(* CoDeSys 2.3 project: WOORI_YANG_BLOCKLIFT_v0.1.pro *)
(* Libraries: INEXT_Library_V01_06.lib 6.7.18 18:58:54, lib_mat.lib 6.7.18 18:58:54, Util.lib 13.6.14 19:20:40, STANDARD_V02_00.lib 6.7.18 18:58:54, BODAS_RC28-14_30_Family_V01_03.lib 6.7.18 18:58:54, CIA405_Library_V02_01.lib 6.7.18 18:58:54, RCE_Library_V01_03.lib 6.7.18 18:58:54, OUTEXT_Library_V01_04.lib 6.7.18 18:58:54, RCE_InitParameter_V01_03.lib 6.7.18 18:58:54, BODAS-design_Library_V20.lib 6.7.18 18:58:54 *)

(* Global variable list: Global_Constant *)
VAR_GLOBAL CONSTANT
	CYCLE_DS16											: INT	  := 20;		(* [ms] main task cycle *)
END_VAR

(* Global variable list: Global_Variables *)
VAR_GLOBAL

	err_s					: applError_ts;		(* BODAS-service error structure, automatically generated by .xls *)
	para_s				: para_ts;				(* BODAS-service parameter structure, automatically generated by .xls *)
	Para					: para_ts;				(* structure for the storage of the parameter *)
	Can		  				: Can_ts;				(* structure for the CAN bus management *)
(*	Err		  				: Error_ts;				(* structure for the error management *) *)
	in_as					: in_as_ts;
(*	Input_raw			: Input_raw_ts;	(* structure for INPUT raw data *) *)
	IO_Chnl				: IO_Chnl_ts; 		(* structure for the channels of the inputs and the outputs *)

END_VAR

(* Data type in Autocode/Enums *)
TYPE applError_e:
(*********************************************)
(*  DON'T MAKE ANY CHANGES TO THIS ENUMS!!   *)
(*     FILE WAS AUTOMATICALLY GENERATED!!    *)
(*********************************************)
(

   ERR_battery_voltage_e                := 16#8000,
   ERR_central_switch_e                 := 16#8001,
   ERR_vss1_5v_e                        := 16#8002,
   ERR_sol1_A_e                         := 16#8003,
   ERR_sol1_B_e                         := 16#8004,
   ERR_can_1_e                          := 16#8005,
   ERR_joy1_ana_e                       := 16#8006

);
END_TYPE

(* Data type in Autocode/Structures *)
TYPE applError_ts:
(***********************************************)
(*  DON'T MAKE ANY CHANGES TO THIS STRUCTURE!! *)
(*      FILE WAS AUTOMATICALLY GENERATED!!     *)
(***********************************************)
STRUCT

   battery_voltage_u8               : BOOL;
   central_switch_u8                : BOOL;
   vss1_5v_u8                       : BOOL;
   sol1_a_u8                        : BOOL;
   sol1_b_u8                        : BOOL;
   can_1_u8                         : BOOL;
   joy1_ana_u8                      : BOOL;

END_STRUCT
END_TYPE

(* Data type in CAN *)
TYPE Can_Box_ts :
STRUCT

(*@CAN*)

(******************************************************************************)
(******************** Definition: databoxes RX  *******************************)
(******************************************************************************)

	Rx_BODAS1		: UINT	:= 2;		(*used BY BODAS Diag*)
	Rx_BODAS2		: UINT	:= 3;		(*used BY BODAS Diag*)
   	Rx_100					: UINT	:= 4;		(*Remote Control Recevier*)
  	Rx_200					: UINT	:= 5;		(*Remote Control Recevier*)
   	Rx_300					: UINT	:= 6;		(*Remote Control Recevier*)
   	Rx_400					: UINT	:= 7;		(*Remote Control Recevier*)

(******************************************************************************)
(******************** Definition: databoxes TX  *******************************)
(******************************************************************************)

	TX_BODAS1		: UINT	:= 1;		(*used BY BODAS Diag*)
	TX_100		: UINT	:= 8;		(*to read status of output*)
	TX_200		: UINT	:= 9;		(*to read status of output*)


END_STRUCT
END_TYPE

(* Data type in CAN *)
TYPE Can_Chnl_ts :
STRUCT

	(* can bus interfaces *)
(*	CANALYZER	: USINT	:= CAN_1;		(* CAN bus used for the communication with BODAS-service*) *)
	CUSTOMER	: USINT	:= CAN_1;		(* CAN bus used by the customer*)

END_STRUCT
END_TYPE

(* Data type in CAN *)
TYPE Can_Data_ts :
STRUCT

	(* @CAN *)
	(* Rx data buffer *)
	regRx_100_au8: 				ARRAY [1..8] OF USINT; 	(* storage of the data from the customer *)
	regRx_200_au8: 				ARRAY [1..8] OF USINT; 	(* storage of the data from the customer *)
	regRx_300_au8: 				ARRAY [1..8] OF USINT; 	(* storage of the data from the customer *)
	regRx_400_au8: 				ARRAY [1..8] OF USINT; 	(* storage of the data from the customer *)

	(* Tx data buffer *)
(*	regTx_CANalyzer1_au8:	ARRAY [1..8] OF USINT; 	(* storage of the data for the diagnostic *)
	regTx_CANalyzer2_au8: 	ARRAY [1..8] OF USINT; 	(* storage of the data for the diagnostic *) *)
	regTx_100_au8: 	ARRAY [1..8] OF USINT; 	(* storage of the data for the customer *)
	regTx_200_au8: 	ARRAY [1..8] OF USINT; 	(* storage of the data for the customer *)


END_STRUCT
END_TYPE

(* Data type in CAN *)
TYPE Can_Id_ts :
STRUCT

(******************************************************************************)
(******************** Definition: CAN IDs  ************************************)
(******************************************************************************)

	RX_100_id:	UINT := 16#1E4;		(* Define receive CAN1 identifier no 4 *)
	RX_200_id: 	UINT := 16#2E4;		(* Define receive CAN1 identifier no 5 *)
	RX_300_id: 	UINT := 16#764;		(* Define receive CAN1 identifier no 6 *)
	RX_400_id: 	UINT := 16#1FF;		(* Define receive CAN1 identifier no 6 *)

	TX_100_id: UDINT := 16#18F001FF;
	TX_200_id: UDINT := 16#18F002FF;


END_STRUCT
END_TYPE

(* Data type in CAN *)
TYPE Can_Status_ts :
STRUCT

(*@CAN*)

	stCAN1_u16		: UINT;

(******************************************************************************)
(******************** Status: databoxes TX  ***********************************)
(******************************************************************************)
(*	stTx_CANalyzer1_u16	: UINT;				(* state of the first databox used for the CAN diagnostic*)
	stTx_CANalyzer2_u16	: UINT;				(* state of the second databox used for the CAN diagnostic*) *)
	stTx_st100_u16	: UINT;				(* state of the databox used to transmit values to the customer*)
	stTx_st200_u16	: UINT;				(* state of the databox used to transmit values to the customer*)

(******************************************************************************)
(******************** Status: databoxes RX  ***********************************)
(******************************************************************************)
	stRx_100_u16	:			UINT;				(*state of the databox used to receive values from the customer*)
	stRx_200_u16	: 			UINT;				(*state of the databox used to receive values from the customer*)
	stRx_300_u16	: 			UINT;				(*state of the databox used to receive values from the customer*)
	stRx_400_u16	: 			UINT;				(*state of the databox used to receive values from the customer*)

END_STRUCT
END_TYPE

(* Data type in CAN *)
TYPE Can_te :
(
	CAN_RESET_STOP_E	 :=0,
	CAN_RESET_START_E	 :=1,
	CAN_RESET_WAIT_E	 :=2
);
END_TYPE

(* Data type in CAN *)
TYPE Can_ts :
STRUCT

	Box: 			CAN_Box_ts;   		(*structure to define the databox-numbers*)
	Id: 				CAN_Id_ts;				(*structure to define the ID *)
	Chnl: 			CAN_Chnl_ts;			(*structure to define the CAN channel used*)
	Data: 			CAN_Data_ts;			(*storage of the data related to the CAN communication*)
	Status: 		CAN_Status_ts;  	(*structure to define the databox-numbers*)

END_STRUCT
END_TYPE

(* Data type in IO *)
TYPE in_as_ts :
STRUCT

	in_as: ARRAY [1..73] OF in_ts;

END_STRUCT
END_TYPE

(* Data type in IO *)
TYPE Input_raw_ts :
STRUCT


(******************************************************************************)
(******************** Definition: Input raw value  ****************************)
(******************************************************************************)

(** Joystick **)
	L1_Joytick_Raw_s32:			DINT;
	L2_Joytick_Raw_s32:			DINT;
	L3_Joytick_Raw_s32:			DINT;
	L4_Joytick_Raw_s32:			DINT;
	M_Joytick_Raw_s32:			DINT;

(** Digital Input **)
	L1_Joy_Up_in_s32: 							DINT;
	L1_Joy_Down_in_s32:						DINT;
	L2_Joy_Up_in_s32: 							DINT;
	L2_Joy_Down_in_s32: 					DINT;
	L3_Joy_Up_in_s32: 							DINT;
	L3_Joy_Down_in_s32: 					DINT;
	L4_Joy_Up_in_s32: 							DINT;
	L4_Joy_Down_in_s32: 					DINT;
	M_Joy_Up_in_s32: 							DINT;
	M_Joy_Down_in_s32: 						DINT;
	Local_L1_Joy_Up_in_s32: 				DINT;
	Local_L1_Joy_Down_in_s32:			DINT;
	Local_L2_Joy_Up_in_s32: 				DINT;
	Local_L2_Joy_Down_in_s32: 		DINT;
	Local_L3_Joy_Up_in_s32: 				DINT;
	Local_L3_Joy_Down_in_s32: 		DINT;
	Local_L4_Joy_Up_in_s32: 				DINT;
	Local_L4_Joy_Down_in_s32: 		DINT;

	Spare1_in_s32:	DINT;
	Spare2_in_s32:	DINT;

END_STRUCT
END_TYPE

(* Data type in IO *)
TYPE IO_Chnl_ts :
STRUCT

(******************************************************************************)
(******************** Definition: Input channel  ****************************)
(******************************************************************************)

(* analog voltage inputs: *)
	AIV_L1_JOYSTICK: 		UDINT	:=	IN_33_AIV;
	AIV_L2_JOYSTICK: 		UDINT	:=	IN_34_AIV;
	AIV_L3_JOYSTICK: 		UDINT	:=	IN_35_AIV;
	AIV_L4_JOYSTICK: 		UDINT	:=	IN_36_AIV;
	AIV_M_JOYSTICK: 		UDINT	:=	IN_37_AIV;

	AIV_SPARE_1:				UDINT  	:=	IN_38_AIV;

(* digital inputs: *)
	AID_L1_JOY_UP: UDINT	:=	IN_1_AID;
	AID_L1_JOY_DN: UDINT	:=	IN_2_AID;
	AID_L2_JOY_UP: 	UDINT	:=	IN_3_AID;
	AID_L2_JOY_DN: UDINT	:=	IN_4_AID;
	AID_L3_JOY_UP: UDINT	:=	IN_5_AID;
	AID_L3_JOY_DN: UDINT	:=	IN_6_AID;
	AID_L4_JOY_UP: UDINT	:=	IN_7_AID;
	AID_L4_JOY_DN: UDINT	:=	IN_8_AID;
	AID_M_JOY_UP: UDINT	:=	IN_9_AID;
	AID_M_JOY_DN: UDINT	:=	IN_10_AID;
	AID_LOCAL_L1_UP: UDINT	:=	IN_11_AID;
	AID_LOCAL_L1_DN: UDINT	:=	IN_12_AID;
	AID_LOCAL_L2_UP: UDINT	:=	IN_13_AID;
	AID_LOCAL_L2_DN: UDINT	:=	IN_14_AID;
	AID_LOCAL_L3_UP: UDINT	:=	IN_15_AID;
	AID_LOCAL_L3_DN: UDINT	:=	IN_16_AID;
	AID_LOCAL_L4_UP: UDINT	:=	IN_17_AID;
	AID_LOCAL_L4_DN: UDINT	:=	IN_18_AID;

	AID_SPARE_2:				UDINT  	:=	IN_19_AID;


(* frequency inputs: *)
(*	DSM_DRIVE:		DWORD	:=	IN_26_DSM; (*EE RC10-10/31*)
	FI_DIESEL:			DWORD	:=	IN_33_FI; (*EE RC10-10/31*) *)

(******************************************************************************)
(******************** Definition: Output channel   *************************)
(******************************************************************************)

(* proportional outputs: *)
	POH_CL_PV1A:	UDINT	:=	OUT_1_POH_CL;
	POH_CL_PV1B:	UDINT	:=	OUT_2_POH_CL;
	POH_CL_PV2A:	UDINT	:=	OUT_3_POH_CL;
	POH_CL_PV2B:	UDINT	:=	OUT_4_POH_CL;
	POH_CL_PV3A:	UDINT	:=	OUT_5_POH_CL;
	POH_CL_PV3B:	UDINT	:=	OUT_6_POH_CL;
	POH_CL_PV4A:	UDINT	:=	OUT_7_POH_CL;
	POH_CL_PV4B:	UDINT	:=	OUT_8_POH_CL;
	POL_CL_PV5A: 	UDINT	:=	OUT_37_POL_CL;
	POL_CL_PV5B:	UDINT	:=	OUT_38_POL_CL;
	POL_CL_PV6A:	UDINT	:=	OUT_39_POL_CL;
	POL_CL_PV6B:	UDINT	:=	OUT_40_POL_CL;
	POL_CL_PV7A:	UDINT	:=	OUT_41_POL_CL;
	POL_CL_PV7B:	UDINT	:=	OUT_42_POL_CL;
	POL_CL_PV8A:	UDINT	:=	OUT_43_POL_CL;
	POL_CL_PV8B:	UDINT	:=	OUT_44_POL_CL;

(* digital outputs: *)
	DOH_PV1AB: UDINT	:=	OUT_21_DOH;
	DOH_PV2AB: UDINT	:=	OUT_22_DOH;
	DOH_PV3AB: UDINT	:=	OUT_23_DOH;
	DOH_PV4AB: UDINT	:=	OUT_24_DOH;
	DOH_PV5AB: UDINT	:=	OUT_25_DOH;
	DOH_PV6AB: UDINT	:=	OUT_26_DOH;
	DOH_PV7AB: UDINT	:=	OUT_27_DOH;
	DOH_PV8AB: UDINT	:=	OUT_28_DOH;

	DOH_SPARE1: UDINT	:=	OUT_19_DOH;
	DOH_SPARE2: UDINT	:=	OUT_20_DOH;

(*
(* switch outputs: *)
	DOH_BRAKE: 		DWORD	:=	OUT_6_DOH;

(* Current*)
	PIC_PUMP: 			DWORD := OUT_1_PIC; (*EE RC10-10/31*)
*)

END_STRUCT
END_TYPE
*)

(* Data type in MAINTASK *)
TYPE MainTaskState_te:
(
	MT_INIT,
	MT_CYCLE
);
END_TYPE

(* Data type in IO *)
TYPE out_as_ts :
STRUCT
	out_as: ARRAY [1..73] OF out_ts;

END_STRUCT
END_TYPE

(* Data type in Autocode/Enums *)
TYPE para_e:
(*********************************************)
(*  DON'T MAKE ANY CHANGES TO THIS ENUMS!!   *)
(*    FILE WAS AUTOMATICALLY GENERATED!!     *)
(*********************************************)
(

(* Input configuration *)

(* Joystick 12 Min Max *)
   EEP_L1_Joy_Up_Min_e                    := 769,      
   EEP_L1_Joy_Up_Max_e                    := 770,      
   EEP_L1_Joy_Down_Min_e                  := 771,      
   EEP_L1_Joy_Down_Max_e                  := 772,      
   EEP_L2_Joy_Up_Min_e                    := 773,      
   EEP_L2_Joy_Up_Max_e                    := 774,      
   EEP_L2_Joy_Down_Min_e                  := 775,      
   EEP_L2_Joy_Down_Max_e                  := 776,      

(* Joystick 34 Min Max *)
   EEP_L3_Joy_Up_Min_e                    := 777,      
   EEP_L3_Joy_Up_Max_e                    := 778,      
   EEP_L3_Joy_Down_Min_e                  := 779,      
   EEP_L3_Joy_Down_Max_e                  := 780,      
   EEP_L4_Joy_Up_Min_e                    := 781,      
   EEP_L4_Joy_Up_Max_e                    := 782,      
   EEP_L4_Joy_Down_Min_e                  := 783,      
   EEP_L4_Joy_Down_Max_e                  := 784,      

(* Joystick Master Min Max *)
   EEP_M_Joy_Up_Min_e                     := 785,      
   EEP_M_Joy_Up_Max_e                     := 786,      
   EEP_M_Joy_Down_Min_e                   := 787,      
   EEP_M_Joy_Down_Max_e                   := 788,      

(* Pump 12 Current Control *)
   EEP_iPump_PV1A_min_e                   := 792,      
   EEP_iPump_PV1A_max_e                   := 793,      
   EEP_iPump_PV1B_min_e                   := 794,      
   EEP_iPump_PV1B_max_e                   := 795,      
   EEP_iPump_PV2A_min_e                   := 796,      
   EEP_iPump_PV2A_max_e                   := 797,      
   EEP_iPump_PV2B_min_e                   := 798,      
   EEP_iPump_PV2B_max_e                   := 799,      

(* Pump 34 Current Control *)
   EEP_iPump_PV3A_min_e                   := 800,      
   EEP_iPump_PV3A_max_e                   := 801,      
   EEP_iPump_PV3B_min_e                   := 802,      
   EEP_iPump_PV3B_max_e                   := 803,      
   EEP_iPump_PV4A_min_e                   := 804,      
   EEP_iPump_PV4A_max_e                   := 805,      
   EEP_iPump_PV4B_min_e                   := 806,      
   EEP_iPump_PV4B_max_e                   := 807,      

(* Pump 56 Current Control *)
   EEP_iPump_PV5A_min_e                   := 808,      
   EEP_iPump_PV5A_max_e                   := 809,      
   EEP_iPump_PV5B_min_e                   := 810,      
   EEP_iPump_PV5B_max_e                   := 811,      
   EEP_iPump_PV6A_min_e                   := 812,      
   EEP_iPump_PV6A_max_e                   := 813,      
   EEP_iPump_PV6B_min_e                   := 814,      
   EEP_iPump_PV6B_max_e                   := 815,      

(* Pump 78 Current Control *)
   EEP_iPump_PV7A_min_e                   := 816,      
   EEP_iPump_PV7A_max_e                   := 817,      
   EEP_iPump_PV7B_min_e                   := 818,      
   EEP_iPump_PV7B_max_e                   := 819,      
   EEP_iPump_PV8A_min_e                   := 820,      
   EEP_iPump_PV8A_max_e                   := 821,      
   EEP_iPump_PV8B_min_e                   := 822,      
   EEP_iPump_PV8B_max_e                   := 823,      

(* Local Pump Current Control *)
   EEP_iPump_Local_PV15A_max_e            := 893,      
   EEP_iPump_Local_PV26A_max_e            := 894,      
   EEP_iPump_Local_PV37A_max_e            := 895,      
   EEP_iPump_Local_PV48A_max_e            := 896,      
   EEP_iPump_Local_PV15B_max_e            := 897,      
   EEP_iPump_Local_PV26B_max_e            := 898,      
   EEP_iPump_Local_PV37B_max_e            := 899,      
   EEP_iPump_Local_PV48B_max_e            := 900,      


(* Input configuration 2 *)

(* Ramp_PV1AB *)
   EEP_Ramp_PV1A_Ascend_e                 := 825,      
   EEP_Ramp_PV1A_Descend_e                := 826,      
   EEP_Ramp_PV1A_Timebase_e               := 827,      
   EEP_Ramp_PV1B_Ascend_e                 := 829,      
   EEP_Ramp_PV1B_Descend_e                := 830,      
   EEP_Ramp_PV1B_Timebase_e               := 831,      

(* Ramp_PV2AB *)
   EEP_Ramp_PV2A_Ascend_e                 := 833,      
   EEP_Ramp_PV2A_Descend_e                := 834,      
   EEP_Ramp_PV2A_Timebase_e               := 835,      
   EEP_Ramp_PV2B_Ascend_e                 := 837,      
   EEP_Ramp_PV2B_Descend_e                := 838,      
   EEP_Ramp_PV2B_Timebase_e               := 839,      

(* Ramp_PV3AB *)
   EEP_Ramp_PV3A_Ascend_e                 := 841,      
   EEP_Ramp_PV3A_Descend_e                := 842,      
   EEP_Ramp_PV3A_Timebase_e               := 843,      
   EEP_Ramp_PV3B_Ascend_e                 := 845,      
   EEP_Ramp_PV3B_Descend_e                := 846,      
   EEP_Ramp_PV3B_Timebase_e               := 847,      

(* Ramp_PV4AB *)
   EEP_Ramp_PV4A_Ascend_e                 := 849,      
   EEP_Ramp_PV4A_Descend_e                := 850,      
   EEP_Ramp_PV4A_Timebase_e               := 851,      
   EEP_Ramp_PV4B_Ascend_e                 := 853,      
   EEP_Ramp_PV4B_Descend_e                := 854,      
   EEP_Ramp_PV4B_Timebase_e               := 855,      

(* Ramp_PV5AB *)
   EEP_Ramp_PV5A_Ascend_e                 := 857,      
   EEP_Ramp_PV5A_Descend_e                := 858,      
   EEP_Ramp_PV5A_Timebase_e               := 859,      
   EEP_Ramp_PV5B_Ascend_e                 := 861,      
   EEP_Ramp_PV5B_Descend_e                := 862,      
   EEP_Ramp_PV5B_Timebase_e               := 863,      

(* Ramp_PV6AB *)
   EEP_Ramp_PV6A_Ascend_e                 := 865,      
   EEP_Ramp_PV6A_Descend_e                := 866,      
   EEP_Ramp_PV6A_Timebase_e               := 867,      
   EEP_Ramp_PV6B_Ascend_e                 := 869,      
   EEP_Ramp_PV6B_Descend_e                := 870,      
   EEP_Ramp_PV6B_Timebase_e               := 871,      

(* Ramp_PV7AB *)
   EEP_Ramp_PV7A_Ascend_e                 := 873,      
   EEP_Ramp_PV7A_Descend_e                := 874,      
   EEP_Ramp_PV7A_Timebase_e               := 875,      
   EEP_Ramp_PV7B_Ascend_e                 := 877,      
   EEP_Ramp_PV7B_Descend_e                := 878,      
   EEP_Ramp_PV7B_Timebase_e               := 879,      

(* Ramp_PV8AB *)
   EEP_Ramp_PV8A_Ascend_e                 := 881,      
   EEP_Ramp_PV8A_Descend_e                := 882,      
   EEP_Ramp_PV8A_Timebase_e               := 883,      
   EEP_Ramp_PV8B_Ascend_e                 := 885,      
   EEP_Ramp_PV8B_Descend_e                := 886,      
   EEP_Ramp_PV8B_Timebase_e               := 887,      


(* Input configuration 3 *)

(* Ramp_PV_Local *)
   EEP_Ramp_PV_Local_Ascend_e             := 889,      
   EEP_Ramp_PV_Local_Descend_e            := 890,      
   EEP_Ramp_PV_Local_Timebase_e           := 891,      

(* AutoLeveling_height *)
   EEP_Max_height_2_e                     := 908,      
   EEP_Max_height_3_e                     := 909,      
   EEP_Max_height_4_e                     := 910,      
   EEP_Min_height_2_e                     := 911,      
   EEP_Min_height_3_e                     := 912,      
   EEP_Min_height_4_e                     := 913,      

(* AutoLeveling_PV *)
   EEP_AutoLeveling_compensator_1_e       := 915,      
   EEP_AutoLeveling_compensator_2_up_e    := 916,      
   EEP_AutoLeveling_compensator_2_down_e  := 917,      
   EEP_AutoLeveling_compensator_3_up_e    := 918,      
   EEP_AutoLeveling_compensator_3_down_e  := 919,      
   EEP_AutoLeveling_compensator_4_up_e    := 920,      
   EEP_AutoLeveling_compensator_4_down_e  := 921,      

(* Distance *)
   EEP_Distance_1_to_4_e                  := 923,      
   EEP_Distance_1_to_2_e                  := 924,      
   EEP_Height_Hysteresis_High_e           := 926,      
   EEP_Height_Hysteresis_Low_e            := 927,      

(* Height_diff_1 *)
   EEP_Height_diff_point_plus_1_e         := 929,      
   EEP_Height_diff_point_plus_2_e         := 930,      
   EEP_Height_diff_point_plus_3_e         := 931,      
   EEP_Height_diff_point_plus_4_e         := 932,      
   EEP_Height_diff_point_plus_5_e         := 933,      
   EEP_Height_diff_point_plus_6_e         := 934,      
   EEP_Height_diff_point_plus_7_e         := 935,      
   EEP_Height_diff_point_plus_8_e         := 936,      

(* Height_diff_2 *)
   EEP_Height_diff_point_minus_1_e        := 938,      
   EEP_Height_diff_point_minus_2_e        := 939,      
   EEP_Height_diff_point_minus_3_e        := 940,      
   EEP_Height_diff_point_minus_4_e        := 941,      
   EEP_Height_diff_point_minus_5_e        := 942,      
   EEP_Height_diff_point_minus_6_e        := 943,      
   EEP_Height_diff_point_minus_7_e        := 944,      
   EEP_Height_diff_point_minus_8_e        := 945,      


(* Distance_diff *)

(* Autoset_Phase *)
   EEP_Autoset_PV_phase_1_e               := 902,      
   EEP_Autoset_PV_phase_2_e               := 903,      
   EEP_Autoset_PV_phase_3_e               := 904,      
   EEP_Autoset_PV_phase_4_e               := 905,      
   EEP_Autoset_PV_phase_5_e               := 906,      
   EEP_AutoLeveling_PV_phase_0_e          := 947,      

(* Autoleveling_Phase_1 *)
   EEP_AutoLeveling_PV_phase_1_e          := 948,      
   EEP_AutoLeveling_PV_phase_2_e          := 949,      
   EEP_AutoLeveling_PV_phase_3_e          := 950,      
   EEP_AutoLeveling_PV_phase_4_e          := 951,      
   EEP_AutoLeveling_PV_phase_5_e          := 952,      
   EEP_AutoLeveling_PV_phase_6_e          := 953,      
   EEP_AutoLeveling_PV_phase_7_e          := 954,      
   EEP_AutoLeveling_PV_phase_8_e          := 955,      

(* Autoleveling_Phase_2 *)
   EEP_AutoLeveling_PV_phase_9_e          := 956,      
   EEP_AutoLeveling_PV_phase_10_e         := 957,      
   EEP_AutoLeveling_PV_phase_11_e         := 958,      
   EEP_AutoLeveling_PV_phase_12_e         := 959,      
   EEP_AutoLeveling_PV_phase_13_e         := 960,      
   EEP_AutoLeveling_PV_phase_14_e         := 961,      
   EEP_AutoLeveling_PV_phase_15_e         := 962,      
   EEP_AutoLeveling_PV_phase_16_e         := 963       

);
END_TYPE

(* Data type in Autocode/Structures *)
TYPE para_ts:
(***********************************************)
(*  DON'T MAKE ANY CHANGES TO THIS STRUCTURE!! *)
(*      FILE WAS AUTOMATICALLY GENERATED!!     *)
(***********************************************)
STRUCT


(* Input configuration *)

(* Joystick 12 Min Max *)
   L1_Joy_Up_Min_s16                  : INT;           (* 2100  (2000 - 3000) *)
   L1_Joy_Up_Max_s16                  : INT;           (* 4500  (4000 - 5000) *)
   L1_Joy_Down_Min_s16                : INT;           (* 2000  (2000 - 3000) *)
   L1_Joy_Down_Max_s16                : INT;           (* 500  (0 - 1000) *)
   L2_Joy_Up_Min_s16                  : INT;           (* 2100  (2000 - 3000) *)
   L2_Joy_Up_Max_s16                  : INT;           (* 4500  (4000 - 5000) *)
   L2_Joy_Down_Min_s16                : INT;           (* 2000  (2000 - 3000) *)
   L2_Joy_Down_Max_s16                : INT;           (* 500  (0 - 1000) *)

(* Joystick 34 Min Max *)
   L3_Joy_Up_Min_s16                  : INT;           (* 2100  (2000 - 3000) *)
   L3_Joy_Up_Max_s16                  : INT;           (* 4500  (4000 - 5000) *)
   L3_Joy_Down_Min_s16                : INT;           (* 2000  (2000 - 3000) *)
   L3_Joy_Down_Max_s16                : INT;           (* 500  (0 - 1000) *)
   L4_Joy_Up_Min_s16                  : INT;           (* 2100  (2000 - 3000) *)
   L4_Joy_Up_Max_s16                  : INT;           (* 4500  (4000 - 5000) *)
   L4_Joy_Down_Min_s16                : INT;           (* 2000  (2000 - 3000) *)
   L4_Joy_Down_Max_s16                : INT;           (* 500  (0 - 1000) *)

(* Joystick Master Min Max *)
   M_Joy_Up_Min_s16                   : INT;           (* 2100  (2000 - 3000) *)
   M_Joy_Up_Max_s16                   : INT;           (* 4500  (4000 - 5000) *)
   M_Joy_Down_Min_s16                 : INT;           (* 2000  (2000 - 3000) *)
   M_Joy_Down_Max_s16                 : INT;           (* 500  (0 - 1000) *)

(* Pump 12 Current Control *)
   iPump_PV1A_min_s16                 : INT;           (* 200  (100 - 300) *)
   iPump_PV1A_max_s16                 : INT;           (* 600  (500 - 700) *)
   iPump_PV1B_min_s16                 : INT;           (* 200  (100 - 300) *)
   iPump_PV1B_max_s16                 : INT;           (* 600  (500 - 700) *)
   iPump_PV2A_min_s16                 : INT;           (* 200  (100 - 300) *)
   iPump_PV2A_max_s16                 : INT;           (* 600  (500 - 700) *)
   iPump_PV2B_min_s16                 : INT;           (* 200  (100 - 300) *)
   iPump_PV2B_max_s16                 : INT;           (* 600  (500 - 700) *)

(* Pump 34 Current Control *)
   iPump_PV3A_min_s16                 : INT;           (* 200  (100 - 300) *)
   iPump_PV3A_max_s16                 : INT;           (* 600  (500 - 700) *)
   iPump_PV3B_min_s16                 : INT;           (* 200  (100 - 300) *)
   iPump_PV3B_max_s16                 : INT;           (* 600  (500 - 700) *)
   iPump_PV4A_min_s16                 : INT;           (* 200  (100 - 300) *)
   iPump_PV4A_max_s16                 : INT;           (* 600  (500 - 700) *)
   iPump_PV4B_min_s16                 : INT;           (* 200  (100 - 300) *)
   iPump_PV4B_max_s16                 : INT;           (* 600  (500 - 700) *)

(* Pump 56 Current Control *)
   iPump_PV5A_min_s16                 : INT;           (* 200  (100 - 300) *)
   iPump_PV5A_max_s16                 : INT;           (* 600  (500 - 700) *)
   iPump_PV5B_min_s16                 : INT;           (* 200  (100 - 300) *)
   iPump_PV5B_max_s16                 : INT;           (* 600  (500 - 700) *)
   iPump_PV6A_min_s16                 : INT;           (* 200  (100 - 300) *)
   iPump_PV6A_max_s16                 : INT;           (* 600  (500 - 700) *)
   iPump_PV6B_min_s16                 : INT;           (* 200  (100 - 300) *)
   iPump_PV6B_max_s16                 : INT;           (* 600  (500 - 700) *)

(* Pump 78 Current Control *)
   iPump_PV7A_min_s16                 : INT;           (* 200  (100 - 300) *)
   iPump_PV7A_max_s16                 : INT;           (* 600  (500 - 700) *)
   iPump_PV7B_min_s16                 : INT;           (* 200  (100 - 300) *)
   iPump_PV7B_max_s16                 : INT;           (* 600  (500 - 700) *)
   iPump_PV8A_min_s16                 : INT;           (* 200  (100 - 300) *)
   iPump_PV8A_max_s16                 : INT;           (* 600  (500 - 700) *)
   iPump_PV8B_min_s16                 : INT;           (* 200  (100 - 300) *)
   iPump_PV8B_max_s16                 : INT;           (* 600  (500 - 700) *)

(* Local Pump Current Control *)
   iPump_Local_PV15A_max_s16          : INT;           (* 600  (100 - 700) *)
   iPump_Local_PV26A_max_s16          : INT;           (* 600  (100 - 700) *)
   iPump_Local_PV37A_max_s16          : INT;           (* 600  (100 - 700) *)
   iPump_Local_PV48A_max_s16          : INT;           (* 600  (100 - 700) *)
   iPump_Local_PV15B_max_s16          : INT;           (* 600  (100 - 700) *)
   iPump_Local_PV26B_max_s16          : INT;           (* 600  (100 - 700) *)
   iPump_Local_PV37B_max_s16          : INT;           (* 600  (100 - 700) *)
   iPump_Local_PV48B_max_s16          : INT;           (* 600  (100 - 700) *)


(* Input configuration 2 *)

(* Ramp_PV1AB *)
   Ramp_PV1A_Ascend_s16               : INT;           (* 400 mA (0 - 1000) *)
   Ramp_PV1A_Descend_s16              : INT;           (* 250 mA (0 - 1000) *)
   Ramp_PV1A_Timebase_s16             : INT;           (* 1000 ms (100 - 3000) *)
   Ramp_PV1B_Ascend_s16               : INT;           (* 400 mA (0 - 1000) *)
   Ramp_PV1B_Descend_s16              : INT;           (* 250 mA (0 - 1000) *)
   Ramp_PV1B_Timebase_s16             : INT;           (* 1000 ms (100 - 3000) *)

(* Ramp_PV2AB *)
   Ramp_PV2A_Ascend_s16               : INT;           (* 400 mA (0 - 1000) *)
   Ramp_PV2A_Descend_s16              : INT;           (* 250 mA (0 - 1000) *)
   Ramp_PV2A_Timebase_s16             : INT;           (* 1000 ms (100 - 3000) *)
   Ramp_PV2B_Ascend_s16               : INT;           (* 400 mA (0 - 1000) *)
   Ramp_PV2B_Descend_s16              : INT;           (* 250 mA (0 - 1000) *)
   Ramp_PV2B_Timebase_s16             : INT;           (* 1000 ms (100 - 3000) *)

(* Ramp_PV3AB *)
   Ramp_PV3A_Ascend_s16               : INT;           (* 400 mA (0 - 1000) *)
   Ramp_PV3A_Descend_s16              : INT;           (* 250 mA (0 - 1000) *)
   Ramp_PV3A_Timebase_s16             : INT;           (* 1000 ms (100 - 3000) *)
   Ramp_PV3B_Ascend_s16               : INT;           (* 400 mA (0 - 1000) *)
   Ramp_PV3B_Descend_s16              : INT;           (* 250 mA (0 - 1000) *)
   Ramp_PV3B_Timebase_s16             : INT;           (* 1000 ms (100 - 3000) *)

(* Ramp_PV4AB *)
   Ramp_PV4A_Ascend_s16               : INT;           (* 400 mA (0 - 1000) *)
   Ramp_PV4A_Descend_s16              : INT;           (* 250 mA (0 - 1000) *)
   Ramp_PV4A_Timebase_s16             : INT;           (* 1000 ms (100 - 3000) *)
   Ramp_PV4B_Ascend_s16               : INT;           (* 400 mA (0 - 1000) *)
   Ramp_PV4B_Descend_s16              : INT;           (* 250 mA (0 - 1000) *)
   Ramp_PV4B_Timebase_s16             : INT;           (* 1000 ms (100 - 3000) *)

(* Ramp_PV5AB *)
   Ramp_PV5A_Ascend_s16               : INT;           (* 400 mA (0 - 1000) *)
   Ramp_PV5A_Descend_s16              : INT;           (* 250 mA (0 - 1000) *)
   Ramp_PV5A_Timebase_s16             : INT;           (* 1000 ms (100 - 3000) *)
   Ramp_PV5B_Ascend_s16               : INT;           (* 400 mA (0 - 1000) *)
   Ramp_PV5B_Descend_s16              : INT;           (* 250 mA (0 - 1000) *)
   Ramp_PV5B_Timebase_s16             : INT;           (* 1000 ms (100 - 3000) *)

(* Ramp_PV6AB *)
   Ramp_PV6A_Ascend_s16               : INT;           (* 400 mA (0 - 1000) *)
   Ramp_PV6A_Descend_s16              : INT;           (* 250 mA (0 - 1000) *)
   Ramp_PV6A_Timebase_s16             : INT;           (* 1000 ms (100 - 3000) *)
   Ramp_PV6B_Ascend_s16               : INT;           (* 400 mA (0 - 1000) *)
   Ramp_PV6B_Descend_s16              : INT;           (* 250 mA (0 - 1000) *)
   Ramp_PV6B_Timebase_s16             : INT;           (* 1000 ms (100 - 3000) *)

(* Ramp_PV7AB *)
   Ramp_PV7A_Ascend_s16               : INT;           (* 400 mA (0 - 1000) *)
   Ramp_PV7A_Descend_s16              : INT;           (* 250 mA (0 - 1000) *)
   Ramp_PV7A_Timebase_s16             : INT;           (* 1000 ms (100 - 3000) *)
   Ramp_PV7B_Ascend_s16               : INT;           (* 400 mA (0 - 1000) *)
   Ramp_PV7B_Descend_s16              : INT;           (* 250 mA (0 - 1000) *)
   Ramp_PV7B_Timebase_s16             : INT;           (* 1000 ms (100 - 3000) *)

(* Ramp_PV8AB *)
   Ramp_PV8A_Ascend_s16               : INT;           (* 400 mA (0 - 1000) *)
   Ramp_PV8A_Descend_s16              : INT;           (* 250 mA (0 - 1000) *)
   Ramp_PV8A_Timebase_s16             : INT;           (* 1000 ms (100 - 3000) *)
   Ramp_PV8B_Ascend_s16               : INT;           (* 400 mA (0 - 1000) *)
   Ramp_PV8B_Descend_s16              : INT;           (* 250 mA (0 - 1000) *)
   Ramp_PV8B_Timebase_s16             : INT;           (* 1000 ms (100 - 3000) *)


(* Input configuration 3 *)

(* Ramp_PV_Local *)
   Ramp_PV_Local_Ascend_s16           : INT;           (* 300 mA (0 - 1000) *)
   Ramp_PV_Local_Descend_s16          : INT;           (* 500 mA (0 - 1000) *)
   Ramp_PV_Local_Timebase_s16         : INT;           (* 1000 ms (100 - 3000) *)

(* AutoLeveling_height *)
   Max_height_2_s16                   : INT;           (* 50 mm (0 - 1000) *)
   Max_height_3_s16                   : INT;           (* 50 mm (0 - 1000) *)
   Max_height_4_s16                   : INT;           (* 50 mm (0 - 1000) *)
   Min_height_2_s16                   : INT;           (* -50 mm (-1000 - 0) *)
   Min_height_3_s16                   : INT;           (* -50 mm (-1000 - 0) *)
   Min_height_4_s16                   : INT;           (* -50 mm (-1000 - 0) *)

(* AutoLeveling_PV *)
   AutoLeveling_compensator_1_s16     : INT;           (* 40 % (0 - 100) *)
   AutoLeveling_compensator_2_up_s16  : INT;           (* 70 % (0 - 100) *)
   AutoLeveling_compensator_2_down_s16: INT;           (* 10 % (0 - 100) *)
   AutoLeveling_compensator_3_up_s16  : INT;           (* 70 % (0 - 100) *)
   AutoLeveling_compensator_3_down_s16: INT;           (* 10 % (0 - 100) *)
   AutoLeveling_compensator_4_up_s16  : INT;           (* 70 % (0 - 100) *)
   AutoLeveling_compensator_4_down_s16: INT;           (* 10 % (0 - 100) *)

(* Distance *)
   Distance_1_to_4_s16                : INT;           (* 485 mm (0 - 10000) *)
   Distance_1_to_2_s16                : INT;           (* 320 mm (0 - 10000) *)
   Height_Hysteresis_High_s16         : INT;           (* 2 mm (0 - 100) *)
   Height_Hysteresis_Low_s16          : INT;           (* 1 mm (0 - 100) *)

(* Height_diff_1 *)
   Height_diff_point_plus_1_s16       : INT;           (* 1 mm (-1000 - 1000) *)
   Height_diff_point_plus_2_s16       : INT;           (* 2 mm (-1000 - 1000) *)
   Height_diff_point_plus_3_s16       : INT;           (* 3 mm (-1000 - 1000) *)
   Height_diff_point_plus_4_s16       : INT;           (* 4 mm (-1000 - 1000) *)
   Height_diff_point_plus_5_s16       : INT;           (* 5 mm (-1000 - 1000) *)
   Height_diff_point_plus_6_s16       : INT;           (* 6 mm (-1000 - 1000) *)
   Height_diff_point_plus_7_s16       : INT;           (* 7 mm (-1000 - 1000) *)
   Height_diff_point_plus_8_s16       : INT;           (* 8 mm (-1000 - 1000) *)

(* Height_diff_2 *)
   Height_diff_point_minus_1_s16      : INT;           (* -1 mm (-1000 - 1000) *)
   Height_diff_point_minus_2_s16      : INT;           (* -2 mm (-1000 - 1000) *)
   Height_diff_point_minus_3_s16      : INT;           (* -3 mm (-1000 - 1000) *)
   Height_diff_point_minus_4_s16      : INT;           (* -4 mm (-1000 - 1000) *)
   Height_diff_point_minus_5_s16      : INT;           (* -5 mm (-1000 - 1000) *)
   Height_diff_point_minus_6_s16      : INT;           (* -6 mm (-1000 - 1000) *)
   Height_diff_point_minus_7_s16      : INT;           (* -7 mm (-1000 - 1000) *)
   Height_diff_point_minus_8_s16      : INT;           (* -8 mm (-1000 - 1000) *)


(* Distance_diff *)

(* Autoset_Phase *)
   Autoset_PV_phase_1_s16             : INT;           (* 100 % (0 - 1000) *)
   Autoset_PV_phase_2_s16             : INT;           (* 70 % (0 - 1000) *)
   Autoset_PV_phase_3_s16             : INT;           (* 50 % (0 - 1000) *)
   Autoset_PV_phase_4_s16             : INT;           (* 30 % (0 - 1000) *)
   Autoset_PV_phase_5_s16             : INT;           (* 10 % (0 - 1000) *)
   AutoLeveling_PV_phase_0_s16        : INT;           (* 40 % (0 - 1000) *)

(* Autoleveling_Phase_1 *)
   AutoLeveling_PV_phase_1_s16        : INT;           (* 1 % (0 - 1000) *)
   AutoLeveling_PV_phase_2_s16        : INT;           (* 5 % (0 - 1000) *)
   AutoLeveling_PV_phase_3_s16        : INT;           (* 10 % (0 - 1000) *)
   AutoLeveling_PV_phase_4_s16        : INT;           (* 20 % (0 - 1000) *)
   AutoLeveling_PV_phase_5_s16        : INT;           (* 28 % (0 - 1000) *)
   AutoLeveling_PV_phase_6_s16        : INT;           (* 33 % (0 - 1000) *)
   AutoLeveling_PV_phase_7_s16        : INT;           (* 36 % (0 - 1000) *)
   AutoLeveling_PV_phase_8_s16        : INT;           (* 38 % (0 - 1000) *)

(* Autoleveling_Phase_2 *)
   AutoLeveling_PV_phase_9_s16        : INT;           (* 42 % (0 - 1000) *)
   AutoLeveling_PV_phase_10_s16       : INT;           (* 44 % (0 - 1000) *)
   AutoLeveling_PV_phase_11_s16       : INT;           (* 47 % (0 - 1000) *)
   AutoLeveling_PV_phase_12_s16       : INT;           (* 52 % (0 - 1000) *)
   AutoLeveling_PV_phase_13_s16       : INT;           (* 60 % (0 - 1000) *)
   AutoLeveling_PV_phase_14_s16       : INT;           (* 70 % (0 - 1000) *)
   AutoLeveling_PV_phase_15_s16       : INT;           (* 75 % (0 - 1000) *)
   AutoLeveling_PV_phase_16_s16       : INT;           (* 80 % (0 - 1000) *)
END_STRUCT
END_TYPE

(* POU PLC_PRG, ST *)
(*************************************************************************************
* Copyright (C)  by WOORI Enterprise, 2020, all rights reserved,
*
*	program:			PLC_PRG
*
*************************************************************************************)

PROGRAM PLC_PRG
VAR

(* program name and version number *)
	stSysInit_u16: 				INT;														          								(* State of Sys_init(...) *)
	SW_Name_as8: 			STRING(32) := 'RC20-10_30_SB_JackUp_v0.1';  			(* Software Name *)
	HW_Name_as8: 			STRING(32) := 'RC30-01D6';													(* Hardware Name *)

(* #### Attention #### : Application only runs on RC28-14/30 only if HW_Name_as8 = 'RC30-00D6' *)
(*
	For other ECUs you have to change the hardware name accordingly:
	'RC30-00D6' for RC28-14/30,
 	'RC30-01D6' for RC20-10/30,
 	'RC30-02D6' for RC12-10/30,
	Remember to choose the appropriate target settings in the resources tab.
*)

(* task definition *)
	stMAIN_Task_u16: 				UINT;			(* State of Sys_registerTask(...), 0 = No Error *)
	MAIN_Task_Handle_u8:		USINT;		(* Task Handler for future reference e.g. checkpoint, duration, ... *)
	stEMCY_u16:         				UINT;

END_VAR

VAR CONSTANT

END_VAR
	(*
	- definition of the SW name
	- definition of the HW name
	- definition of a main task   
	- definition of a 'callback' function for the reading of the parameters
	- reading of all parameters
	- configuration of the sensor supply
	- initialisation of the CAN communication
	- initialisation of the input signals 
	- initialisation of the output signals
	*******************************************************************************)

	(* mandatory *)
	(******************************************************************************)
	(******************* definition: SW name and HW name **************************)
	(******************************************************************************)
	stSysInit_u16 := sys_init(ADR(SW_Name_as8), ADR(HW_Name_as8));
	(* sys_init() : This function initializes the system *)

	(* mandatory *)
	(******************************************************************************)
	(******************** definition: main task   **************************************)
	(******************************************************************************)
	stMAIN_Task_u16 := sys_registerTask(
																				func_pf:=	INDEXOF(_0_Callback_MAIN_Task),
																				priority_u8:= 60,
																				cycleTime_ms_u32:= 20,
																				cycleOffset_ms_u32:= 0,
																				taskHandle_pu8:=	 ADR(MAIN_Task_Handle_u8));

	(* Set trigger checkpoint for above task *)
	sys_initTC(checkPoint_u8:= MAIN_Task_Handle_u8, interval_u8:= 20);

	(* mandatory *)
	(******************************************************************************)
	(****************** definition: callback to load the parameters****************)
	(******************************************************************************)

	(* register callback function for parameters *)
	diag_setVarsCallBack(INDEXOF(Callback_diag_getPara));
	(* The application uses the function diag_setVarsCallBack() to declare a copy function with the system that copies application data from the EEPROM to the application variables *)

	(* load all parameters when starting up *)
	Callback_diag_getPara();

	(******************************************************************************)
	(******************** Configuration: Input  ***********************************)
	(******************************************************************************)
	PLC_cfgInputs();

	(******************************************************************************)
	(******************** Configuration:Outputs *********************************)
	(******************************************************************************)
	PLC_cfgOutputs();
(*	PLC_cfgOutputs_LAB(); *)

	(******************************************************************************)
	(********************* Initialization: CAN communication  *********************)
	(******************************************************************************)
	PLC_initCAN();

	(* necessary if just TB3 with Low channel is used *)
	(* disable the software INHIBIT *)
	(* This command is necessary if pin 112 shall be used as input and not as software INH input *)
	stEMCY_u16 := emcy_disableInput(EMCY_DISABLE_KEY_DU32, NOT UDINT_TO_DWORD(EMCY_DISABLE_KEY_DU32));
END_PROGRAM
ACTION ChangeRequestHistory:
;

(*

	2023.05.26.		|		creat 				|	v0.1 

*)
END_ACTION
ACTION PLC_cfgInputs:
(*------------------------------------------------------------------------------ VSS Configure ------------------------------------------------------------------------------*)
	(* at RC28-14 is VSS1 always ON *)
	(* switch on VSS_2 and VSS_3 sensor supply *)
	sys_setVSS(VSS_2, ON);		(* 10V @ RC28-14 *)
	sys_setVSS(VSS_3, ON);		(*  5V @ RC28-14 *)

(*------------------------------------------------------------------------------ Current Configure ------------------------------------------------------------------------------*)

	(* switch on shunt for pin138: group1:  IN_52_AIC *)
	(*		Group 1:	IN_52,  IN_53
    		Group 2:	IN_54,  IN_55,  IN_56,  IN_57	 
    		Group 3: 	IN_58,  IN_59,  IN_60,  IN_61
			in_setCurrentMeasurement(group, state_I); 	state_I => ON - current/ OFF - voltage *)

	in_setCurrentMeasurement(1, ON);
(*	in_setCurrentMeasurement(2, ON);
	in_setCurrentMeasurement(3, ON); *)

(*------------------------------------------------------------------------------ Analog Input ------------------------------------------------------------------------------*)

	in_cfgCurrentInput(IN_52_AIC, 200);		(* GEFRAN distance X sensor *)
	in_cfgCurrentInput(IN_53_AIC, 200);		(* GEFRAN distance Y sensor *)
	in_cfgCurrentInput(IN_54_AIC, 200);		(* GEFRAN distance Z sensor *)

(*	in_cfgCurrentInput(IN_56_AIC, 200);		(* Current-meter from Control Panel *) *)

	in_cfgVoltageInput(IN_55_AIV,	2000,	3000, 100, 1500, 3500, 200);		(* Volt-meter from Control Panel *)

	in_cfgVoltageInput(IN_1_AIV,	2000,	3000, 100, 1500, 3500, 200);			(* GEFRAN pressure sensor of  X - A *)
	in_cfgVoltageInput(IN_2_AIV,	2000,	3000, 100, 1500, 3500, 200);			(* GEFRAN pressure sensor of  X - B *)
	in_cfgVoltageInput(IN_3_AIV,	2000,	3000, 100, 1500, 3500, 200);			(* GEFRAN pressure sensor of  Y - A *)
	in_cfgVoltageInput(IN_4_AIV,	2000,	3000, 100, 1500, 3500, 200);			(* GEFRAN pressure sensor of  Y - B *)
	in_cfgVoltageInput(IN_5_AIV,	2000,	3000, 100, 1500, 3500, 200);			(* GEFRAN pressure sensor of  Z - A *)
	in_cfgVoltageInput(IN_6_AIV,	2000,	3000, 100, 1500, 3500, 200);			(* GEFRAN pressure sensor of  Z - B *)
	in_cfgVoltageInput(IN_7_AIV,	2000,	3000, 100, 1500, 3500, 200);			(* GEFRAN pressure sensor of Main System *)

	in_cfgVoltageInput(IN_8_AIV,	2000,	3000, 100, 1500, 3500, 200);			(* Track Joystick from Handle Bar *)

	in_cfgTempSensorType(IN_62_AIT, 255);														(* Temperature Sensor *)

(*------------------------------------------------------------------------------ Digital Input ------------------------------------------------------------------------------*)

	in_cfgVoltageInput(IN_9_AID, 5000, 8000, 200, 1500, 10000, 200); 		(* EMERGENCY from Control Panel - Digital Input *)
	in_cfgVoltageInput(IN_10_AID, 5000, 8000, 200, 1500, 10000, 200); 		(* REMOTE SELECT from Control Panel - Digital Input *)
	in_cfgVoltageInput(IN_11_AID,	5000, 8000, 200, 1500, 10000, 200); 		(* MANUAL SELECT from Control Panel - Digital Input *)
	in_cfgVoltageInput(IN_12_AID, 5000, 8000, 200, 1500, 10000, 200);		(* HEATER ON from Control Panel - Digital Input *)
	in_cfgVoltageInput(IN_13_AID, 5000, 8000, 200, 1500, 10000, 200); 		(* ENGINE ON from Control Panel - Digital Input *)
	in_cfgVoltageInput(IN_14_AID, 5000, 8000, 200, 1500, 10000, 200);		(* ENGINE OFF from Control Panel - Digital Input *)
	in_cfgVoltageInput(IN_15_AID, 5000, 8000, 200, 1500, 10000, 200); 		(* WHEEL UP from Control Panel - Digital Input *)
	in_cfgVoltageInput(IN_16_AID, 5000, 8000, 200, 1500, 10000, 200); 		(* WHEEL DOWN from Control Panel - Digital Input *)
	in_cfgVoltageInput(IN_17_AID, 5000, 8000, 200, 1500, 10000, 200); 		(* BUZZER ON from Control Panel - Digital Input *)
	in_cfgVoltageInput(IN_18_AID, 5000, 8000, 200, 1500, 10000, 200); 		(* ALARM OFF from Control Panel - Digital Input *)
	in_cfgVoltageInput(IN_19_AID, 5000, 8000, 200, 1500, 10000, 200);		(* CYL Z UP from Control Panel - Digital Input *)
	in_cfgVoltageInput(IN_20_AID, 5000, 8000, 200, 1500, 10000, 200); 		(* CYL Z DOWN from Control Panel - Digital Input *)
	in_cfgVoltageInput(IN_21_AID, 5000, 8000, 200, 1500, 10000, 200); 		(* CYL X, Y EXTEND from Control Panel - Digital Input *)
	in_cfgVoltageInput(IN_22_AID, 5000, 8000, 200, 1500, 10000, 200);		(* CYL X, Y EXTRACT from Control Panel - Digital Input *)
	in_cfgVoltageInput(IN_23_AID, 5000, 8000, 200, 1500, 10000, 200); 		(* CYL X SELECT from Control Panel - Digital Input *)
	in_cfgVoltageInput(IN_24_AID, 5000, 8000, 200, 1500, 10000, 200); 		(* CYL Y SELECT from Control Panel - Digital Input *)
	in_cfgVoltageInput(IN_25_AID, 5000, 8000, 200, 1500, 10000, 200);		(* Wheel Rest Proximity Sensor 1 from Control Panel - Digital Input *)
	in_cfgVoltageInput(IN_26_AID, 5000, 8000, 200, 1500, 10000, 200); 		(* Wheel Rest Proximity Sensor 2 from Control Panel - Digital Input *)
	in_cfgVoltageInput(IN_27_AID, 5000, 8000, 200, 1500, 10000, 200);		(* Wheel Rest Proximity Sensor 3 from Control Panel - Digital Input *)
	in_cfgVoltageInput(IN_28_AID, 5000, 8000, 200, 1500, 10000, 200); 		(* ZERO RETURN from Control Panel - Digital Input *)
	in_cfgVoltageInput(IN_29_AID, 5000,	8000, 200, 1500, 10000, 200); 		(* Oil Level Low Swith from Oil Tank - Digital Input *)
	in_cfgVoltageInput(IN_30_AID, 5000,	8000, 200, 1500, 10000, 200); 		(* Oil Level Low-Low Swith from Oil Tank - Digital Input *)
	in_cfgVoltageInput(IN_31_AID, 5000, 8000, 200, 1500, 10000, 200); 		(* Oil Filter Indicator from Water Seperator- Digital Input *)
(*	in_cfgVoltageInput(IN_32_AID, 5000,	8000, 200, 1500, 10000, 200); 		(* Oil Temperature High from Oil Tank - Digital Input *) *)
	in_cfgVoltageInput(IN_33_AID, 5000,	8000, 200, 1500, 10000, 200); 		(* Overcurrent from Control Panel - Digital Input*)

	in_cfgVoltageInput(IN_43_DI, 5000,	8000, 200, 1500, 10000, 200); 			(* Select A from Control Panel - Digital Input*)
	in_cfgVoltageInput(IN_44_DI, 5000,	8000, 200, 1500, 10000, 200); 			(* Select B from Control Panel - Digital Input*)
	in_cfgVoltageInput(IN_45_DI, 5000,	8000, 200, 1500, 10000, 200); 			(* Select C from Control Panel - Digital Input*)
	in_cfgVoltageInput(IN_46_DI, 5000,	8000, 200, 1500, 10000, 200); 			(* Select D from Control Panel - Digital Input*)
	in_cfgVoltageInput(IN_47_DI, 5000,	8000, 200, 1500, 10000, 200); 			(* Select Group 1 from Control Panel - Digital Input*)
	in_cfgVoltageInput(IN_48_DI, 5000,	8000, 200, 1500, 10000, 200); 			(* Select Group 2 from Control Panel - Digital Input*)

(*------------------------------------------------------------------------------ Spare Input ------------------------------------------------------------------------------*)

	in_cfgVoltageInput(IN_34_AIV,	2000,	3000, 100, 1500, 3500, 200);		(* Spare Analog Input *)
	in_cfgVoltageInput(IN_35_AIV,	2000,	3000, 100, 1500, 3500, 200);		(* Spare Analog Input *)
	in_cfgVoltageInput(IN_36_AIV,	2000,	3000, 100, 1500, 3500, 200);		(* Spare Analog Input *)
	in_cfgVoltageInput(IN_37_AIV,	2000,	3000, 100, 1500, 3500, 200);		(* Spare Analog Input *)
	in_cfgVoltageInput(IN_38_AIV,	2000,	3000, 100, 1500, 3500, 200);		(* Spare Analog Input *)


   (* 이 함수를 사용하는 채널들은 uUpperDiagThreshold_u16값을 최대 10V까지만 사용해야 한다. Datasheet 11page 참조. IN *)
	(* IN_1 ~ IN_24, IN_25 ~ IN_32, IN_40 ~ IN_41 까지의 Analog와  Digital 입력을 공용으로 사용하는 입력 채널 ~!!! *)
	(* signal debounce time, default 100ms, 토글스위치의 경우 이값을 최소 200 조정 필요함~~!!! 100인경우 채터링으로 인해 입력이 튕겨져 나옴.  *)
(*
	in_cfgDigitalInput(IN_43_DI, 200); (* IN42~51까지만 사용할 수 있는 펑션임. *)
	(* 내부 Pull-up 저항때문에 이 채널 IN_43 ~ IN_51까지는 GND를 연결해야 Toggle Switch 입력으로 사용할 수 있다. !!! *)

	(* Config current input EXAMPLE *)
	in_cfgCurrentInput(IN_52_AIC, 200);
*)
END_ACTION
ACTION PLC_cfgOutputs:
(*------------------------------------------------------------------------------ Propotional Valve Configuration ------------------------------------------------------------------------------*)

		(** OUT_1  for CYL X UP  **)
		out_cfg(OUT_1_POH_CL,100, tiPeriod_10ms_DU16, 14700, 43400);
(*		out_cfgDither(OUT_1_POH_CL, fDither_100Hz_DU8, 200 ); *)
		out_cfgPI(OUT_1_POH_CL, 367, 262);
		out_cfgSlope(OUT_1_POH_CL, 2000);

		(** OUT_2  for CYL X DOWN  **)
		out_cfg(OUT_2_POH_CL,100, tiPeriod_10ms_DU16, 14700, 43400);
(*		out_cfgDither(OUT_2_POH_CL, fDither_100Hz_DU8, 200 ); *)
		out_cfgPI(OUT_2_POH_CL, 367, 262);
		out_cfgSlope(OUT_2_POH_CL, 2000);

		(** OUT_3  for CYL Y UP **)
		out_cfg(OUT_3_POH_CL,100, tiPeriod_10ms_DU16, 14700, 43400);
(*		out_cfgDither(OUT_3_POH_CL, fDither_100Hz_DU8, 200 ); *)
		out_cfgPI(OUT_3_POH_CL, 367, 262);
		out_cfgSlope(OUT_3_POH_CL, 2000);

		(** OUT_4  for CYL Y DOWN **)
		out_cfg(OUT_4_POH_CL,100, tiPeriod_10ms_DU16, 14700, 43400);
(*		out_cfgDither(OUT_4_POH_CL, fDither_100Hz_DU8, 200 ); *)
		out_cfgPI(OUT_4_POH_CL, 367, 262);
		out_cfgSlope(OUT_4_POH_CL, 2000);

		(** OUT_5  for CYL Z (no-load) UP **)
		out_cfg(OUT_5_POH_CL,100, tiPeriod_10ms_DU16, 14700, 43400);
(*		out_cfgDither(OUT_5_POH_CL, fDither_100Hz_DU8, 200 ); *)
		out_cfgPI(OUT_5_POH_CL, 367, 262);
		out_cfgSlope(OUT_5_POH_CL, 2000);

		(** OUT_6  for CYL Z (no-load) DOWN  **)
		out_cfg(OUT_6_POH_CL,100, tiPeriod_10ms_DU16, 14700, 43400);
(*		out_cfgDither(OUT_6_POH_CL, fDither_100Hz_DU8, 200 ); *)
		out_cfgPI(OUT_6_POH_CL, 367, 262);
		out_cfgSlope(OUT_6_POH_CL, 2000);

		(** OUT_7  for CYL Z (load) UP **)
		out_cfg(OUT_7_POH_CL,100, tiPeriod_10ms_DU16, 14700, 43400);
(*		out_cfgDither(OUT_7_POH_CL, fDither_100Hz_DU8, 200 ); *)
		out_cfgPI(OUT_7_POH_CL, 367, 262);
		out_cfgSlope(OUT_7_POH_CL, 2000);

		(** OUT_8  for CYL Z (load) DOWN **)
		out_cfg(OUT_8_POH_CL,100, tiPeriod_10ms_DU16, 14700, 43400);
(*		out_cfgDither(OUT_8_POH_CL, fDither_100Hz_DU8, 200 ); *)
		out_cfgPI(OUT_8_POH_CL, 367, 262);
		out_cfgSlope(OUT_8_POH_CL, 2000);

		(** OUT_9  for WHEEL FORWARD **)
		out_cfg(OUT_9_POH_CL,100, tiPeriod_10ms_DU16, 14700, 43400);
(*		out_cfgDither(OUT_9_POH_CL, fDither_100Hz_DU8, 200 ); *)
		out_cfgPI(OUT_9_POH_CL, 367, 262);
		out_cfgSlope(OUT_9_POH_CL, 2000);

		(** OUT_10  for WHEEL BACKWARD **)
		out_cfg(OUT_10_POH_CL,100, tiPeriod_10ms_DU16, 14700, 43400);
(*		out_cfgDither(OUT_10_POH_CL, fDither_100Hz_DU8, 200 ); *)
		out_cfgPI(OUT_10_POH_CL, 367, 262);
		out_cfgSlope(OUT_10_POH_CL, 2000);

		(** OUT_37  for WHEEL UP **)
		out_cfg(OUT_37_POL_CL,100, tiPeriod_10ms_DU16, 14700, 43400);
(*		out_cfgDither(OUT_37_POL_CL, fDither_100Hz_DU8, 200 ); *)
		out_cfgPI(OUT_37_POL_CL,500, 357);
		out_cfgSlope(OUT_37_POL_CL, 2000);

		(** OUT_38  for WHEEL DOWN **)
		out_cfg(OUT_38_POL_CL,100, tiPeriod_10ms_DU16, 14700, 43400);
(*		out_cfgDither(OUT_38_POL_CL, fDither_100Hz_DU8, 200 ); *)
		out_cfgPI(OUT_38_POL_CL, 367, 262);
		out_cfgSlope(OUT_38_POL_CL, 2000);

(*------------------------------------------------------------------------------ Digital Output Configuration ------------------------------------------------------------------------------*)

		(* OUT_19  for 3-WAY sol-valve *)
		out_cfg(
						chnl_u32								:= OUT_19_DOH,							(* Channel number: PWM highside output close loop *)
						tiDiagDebounce_u16			:= 100,												(* debounce time [ms] for error detection *)
						freq_u16								:= tiPeriod_10ms_DU16,				(* 100Hz repetition time [ms] = 1 / dither frequency *)
						rMinLoad_u32						:= 3000,												(* min resistance of solenoid for error detection [mOhm] *)
						rMaxLoad_u32						:= 9000);											(* max resistance of solenoid for error detection[mOhm] *)

		out_cfg(OUT_20_DOH, 100, tiPeriod_10ms_DU16, 3000, 9000);		(* OUT_20 for Unloading sol-valve *)
		out_cfg(OUT_21_DOH, 100, tiPeriod_10ms_DU16, 3000, 9000);		(* BUZZER ON - Digital Output *)
		out_cfg(OUT_22_DOH, 100, tiPeriod_10ms_DU16, 3000, 9000);		(* Engine Start - Digital Output *)
		out_cfg(OUT_23_DOH, 100, tiPeriod_10ms_DU16, 3000, 9000);		(* Engine Stop - Digital Output *)
		out_cfg(OUT_24_DOH, 100, tiPeriod_10ms_DU16, 3000, 9000);		(* HEATER ON - Digital Output *)
		out_cfg(OUT_25_DOH, 100, tiPeriod_10ms_DU16, 3000, 9000);		(* Termination Resistance ON/OFF - Digital Output *)
END_ACTION
ACTION PLC_initCAN:
(*------------------------------------------------------------------------------ CAN initiation ------------------------------------------------------------------------------*)

can_init(CAN_1, BAUD_250K);
(* can_init(CAN_2, BAUD_250K); *)
(* can_init(CAN_3, BAUD_250K); *)
(* can_init(CAN_4, BAUD_250K); *)

(*------------------------------------------------------------------------------ CAN receive message ------------------------------------------------------------------------------*)
(* !: databox numbers 2 + 3 are reserved and already used by B-d communication ! *)

can_cfgRxDatabox(CAN.Chnl.CUSTOMER,  		(* chnl_u8 *)
                 			    	CAN.Box.RX_100,   				(* databoxNum_s16 *)
					             	CAN.Id.RX_100_id,    				(* id_u32 *)
					             	CAN_STD_DU8);    	   			(* format_u8 *)

can_cfgRxDatabox(CAN.Chnl.CUSTOMER,  		(* chnl_u8 *)
                 				 	CAN.Box.RX_200,   				(* databoxNum_s16 *)
					             	CAN.Id.RX_200_id,    				(* id_u32 *)
					             	CAN_STD_DU8);       				(* format_u8 *)

can_cfgRxDatabox(CAN.Chnl.CUSTOMER,  		(* chnl_u8 *)
                 				 	CAN.Box.RX_300,   				(* databoxNum_s16 *)
					             	CAN.Id.RX_300_id,    				(* id_u32 *)
					             	CAN_STD_DU8);       				(* format_u8 *)

can_cfgRxDatabox(CAN.Chnl.CUSTOMER,  		(* chnl_u8 *)
                 				 	CAN.Box.RX_400,   				(* databoxNum_s16 *)
					             	CAN.Id.RX_400_id,    				(* id_u32 *)
					             	CAN_STD_DU8);       				(* format_u8 *)

(*------------------------------------------------------------------------------ CAN transmit message ------------------------------------------------------------------------------*)
(* !: databox number 1 is reserved and already used by B-d communication ! *)

can_cfgTxDatabox(CAN.Chnl.CUSTOMER,			(* chnl_u8 *)
						     		CAN.Box.TX_100,  		(* databoxNum_s16 *)
						     		CAN.Id.TX_100_id,	 	(* id_u32 *)
						     		CAN_EXD_DU8);					(* format_u8 *)

can_cfgTxDatabox(CAN.Chnl.CUSTOMER,			(* chnl_u8 *)
						     		CAN.Box.TX_200,  		(* databoxNum_s16 *)
						     		CAN.Id.TX_200_id,	 	(* id_u32 *)
						     		CAN_EXD_DU8);					(* format_u8 *)
END_ACTION

(* POU _0_Callback_MAIN_Task, ST *)
PROGRAM _0_Callback_MAIN_Task
VAR

(**** 01_INIT ****)

	setVP_1: INT; 							(* state of the power supply1 *)
	setVP_2: UINT; 						(* state of the power supply2 *)

	stSupplyVP1_b: BOOL;			(*state of the supply VP1*)
	stSupplyVP2_b: BOOL;			(*state of the supply VP2*)

	Voltage_VSS_1: UINT; 			(* Supply Voltage VSS_1 *)
	Voltage_VSS_2: UINT; 			(* Supply Voltage VSS_2 *)
	Voltage_VSS_3: UINT; 			(* Supply Voltage VSS_ 3*)

	Voltage_VP_1: UINT; 				(* Supply Voltage VP_1 *)
	Voltage_VP_2: UINT; 				(* Supply Voltage VP_2 *)

	stSysEMCY_b: BOOL; 			(*State of the emergency switch*)
	stSysINH_b: BOOL;					(*State of INH (pin228)*)
	tiSysRunTime_s32: DINT;		(*duration of the task*)
	etaSysTaskLoad_s16: INT;		(*load of the main task*)

	STARTLOCK_Condition: INT;
	Start_State: BOOL;

	TON_Init: TON;

END_VAR

VAR CONSTANT
	DELAY_STANDARD : INT  := 500;		(* debouncing time 500[ms] *)
	ERR_0 : BYTE := 0;		(* error no for B-s text inputs *)
	STARTLOCK_Check_Supply_VB : INT	:= 0;
	STARTLOCK_Check_Supply_VSS : INT	:= 1;
	STARTLOCK_RUN : INT 	:= 2;
	STARTLOCK_ERROR : INT 	:= 3;
END_VAR

VAR_INPUT
END_VAR
(* trigger checkpoint, mandatory *)
sys_triggerTC(PLC_PRG.MAIN_Task_Handle_u8);

setVP_1 := sys_setVP(VP_1, ON); (* PWM-supply *)
setVP_2 := sys_setVP(VP_2, ON); (* DIGout-supply *)

stSupplyVP1_b	:= sys_getVP(VP_1); (* State of the supply VP1 *)
stSupplyVP2_b	:= sys_getVP(VP_2); (* State of the supply VP2 *)

Voltage_VSS_1	:= sys_getSupply(VSS_1);
Voltage_VSS_2	:= sys_getSupply(VSS_2);
Voltage_VSS_3	:= sys_getSupply(VSS_3);

Voltage_VP_1		:= sys_getSupply(VP_1);
Voltage_VP_2		:= sys_getSupply(VP_2);

(*check the state OF 'INH': excepted value: OFF*)
stSysINH_b			:= USINT_TO_BOOL(sys_getINH( ));
stSysEMCY_b	:= emcy_getStatus( );

tiSysRunTime_s32 		:= sys_getTaskRunTime(PLC_PRG.MAIN_Task_Handle_u8, PTIME_AVERAGE_INCL);
etaSysTaskLoad_s16 	:= sys_getTaskLoad(PTIME_AVERAGE_INCL);


CASE STARTLOCK_Condition OF

(*0- check Vb supply > 8.5V*)
STARTLOCK_Check_Supply_VB:
		(* startcondition flag *)
		Start_State	:= FALSE;
		(* transition *)
 		IF (Voltage_VP_1 > 8500) THEN
			STARTLOCK_Condition := STARTLOCK_Check_Supply_VSS;
		END_IF

(*1- check Vssx > threshold*)
STARTLOCK_Check_Supply_VSS:
		(* startcondition flag *)
		Start_State	:= FALSE;
		(* transition *)
	(*	IF ( *)
	(*		(uSupply_VSS_1_mV_u16 > 4500) AND *) (* EE RC10-10/31 could not be measured*)
	(*		(uSupply_VSS_2_mV_u16 > 9500) AND *) (* EE RC10-10/31 not switched on without load *)
	(*		(uSupply_VSS_3_mV_u16 > 4500)   *)   (* EE RC10-10/31 could not be measured*)
	(*		) THEN *)
		STARTLOCK_Condition	:= STARTLOCK_RUN;
	(*	ELSE
			;           
		END_IF *)

(*2- RUN *)
STARTLOCK_RUN:
		(* startcondition flag *)
		Start_State	:= TRUE;
		(* transition *)
		STARTLOCK_Condition	:= STARTLOCK_RUN;

ELSE
	(* this state should never be reached *)
	STARTLOCK_Condition := STARTLOCK_Check_Supply_VSS;

END_CASE

TON_Init(in := TRUE, PT := T#1000ms);

IF Start_State AND TON_Init.Q THEN

	_1_CAN_IN();
	_2_IN_RC();
	_3_RUN();
	_4_PROCESS_VALUES();
	_5_OUT_RC();

END_IF;
END_PROGRAM

(* POU _1_CAN_IN, FBD *)
PROGRAM _1_CAN_IN
VAR

	(* Wireless *)
	can_in_wireless_Left_Joy : INT;
	can_in_wireless_Right_Joy : INT;

	(* Wire *)
	can_in_wire_Left_Joy: INT;
	can_in_wire_Right_Joy: INT;

	(* CANlink_4000 *)

	(* CANlink_3000 *)

END_VAR
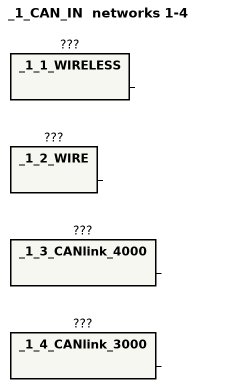
_FBD_ (* Function Block Diagram *)
NETWORK 1
	???:_1_1_WIRELESS()
NETWORK 2
	???:_1_2_WIRE()
NETWORK 3
	???:_1_3_CANlink_4000()
NETWORK 4
	???:_1_4_CANlink_3000()
_END_FBD_
END_PROGRAM
ACTION _1_1_WIRELESS:
;
END_ACTION
ACTION _1_2_WIRE:
;
END_ACTION
ACTION _1_3_CANlink_4000:
;
END_ACTION
ACTION _1_4_CANlink_3000:
;
END_ACTION

(* POU _2_IN_RC, ST *)
PROGRAM _2_IN_RC
VAR

	in_as: ARRAY [1..73] OF in_ts;

(* _2_1_Panel *)

	in_Panel_Emegency: BOOL;
	in_Panel_Wireless: BOOL;
	in_Panel_Wire: BOOL;
	in_Panel_Manual: BOOL;
	in_Panel_Heater: BOOL;
	in_Panel_Engine_On: BOOL;
	in_Panel_Engine_Off: BOOL;
	in_Panel_Wheel_Up: BOOL;
	in_Panel_Wheel_Down: BOOL;
	in_Panel_Buzzer_On: BOOL;
	in_Panel_Buzzer_Off: BOOL;
	in_Panel_Cyl_Z_Up: BOOL;
	in_Panel_Cyl_Z_Down: BOOL;
	in_Panel_Cyl_XY_Up: BOOL;
	in_Panel_Cyl_XY_Down: BOOL;
	in_Panel_X_select: BOOL;
	in_Panel_Y_select: BOOL;
	in_Panel_Zero_Return: BOOL;
	in_Panel_A_select: BOOL;
	in_Panel_B_select: BOOL;
	in_Panel_C_select: BOOL;
	in_Panel_D_select: BOOL;
	in_Panel_Group1_select: BOOL;
	in_Panel_Group2_select: BOOL;
	in_Panel_Voltmeter: INT;

(* _2_2_HANDELBAR *)

	in_Handlebar_Joy: DINT;

(* _2_2_HANDLEBAR *)

	Handelbar_Joy_upward: DINT;
	Handelbar_Joy_downward: DINT;

(* _2_3_SENSORS *)

	in_Sensor_Distance_X: INT;
	in_Sensor_Distance_Y: INT;
	in_Sensor_Distance_Z: INT;
	in_Sensor_Voltage: INT;
	in_Sensor_Pressure_X_A: INT;
	in_Sensor_Pressure_X_B: INT;
	in_Sensor_Pressure_Y_A: INT;
	in_Sensor_Pressure_Y_B: INT;
	in_Sensor_Pressure_Z_A: INT;
	in_Sensor_Pressure_Z_B: INT;
	in_Sensor_Pressure_Main: INT;
	in_Sensor_Temp: INT;
	in_Sensor_Wheel_rest: BOOL;
	in_Sensor_Oil_Low: BOOL;
	in_Sensor_Oil_Low_Low: BOOL;
	in_Sensor_Filter_indicator: BOOL;
	in_Sensor_Temp_High: BOOL;
	in_Sensor_Overcurrent: BOOL;


END_VAR
(*------------------------------------------------------------------------------ INXT ------------------------------------------------------------------------------*)

	inxt(IN_1_AIV, ADR(in_as[1]));
	inxt(IN_2_AIV, ADR(in_as[2]));
	inxt(IN_3_AIV, ADR(in_as[3]));
	inxt(IN_4_AIV, ADR(in_as[4]));
	inxt(IN_5_AIV, ADR(in_as[5]));
	inxt(IN_6_AIV, ADR(in_as[6]));
	inxt(IN_7_AIV, ADR(in_as[7]));
	inxt(IN_8_AIV, ADR(in_as[8]));
	inxt(IN_9_AID, ADR(in_as[9]));
	inxt(IN_10_AID, ADR(in_as[10]));
	inxt(IN_11_AID, ADR(in_as[11]));
	inxt(IN_12_AID, ADR(in_as[12]));
	inxt(IN_13_AID, ADR(in_as[13]));
	inxt(IN_14_AID, ADR(in_as[14]));
	inxt(IN_15_AID, ADR(in_as[15]));
	inxt(IN_16_AID, ADR(in_as[16]));
	inxt(IN_17_AID, ADR(in_as[17]));
	inxt(IN_18_AID, ADR(in_as[18]));
	inxt(IN_19_AID, ADR(in_as[19]));
	inxt(IN_20_AID, ADR(in_as[20]));
	inxt(IN_21_AID, ADR(in_as[21]));
	inxt(IN_22_AID, ADR(in_as[22]));
	inxt(IN_23_AID, ADR(in_as[23]));
	inxt(IN_24_AID, ADR(in_as[24]));
	inxt(IN_25_AID, ADR(in_as[25]));
	inxt(IN_26_AID, ADR(in_as[26]));
	inxt(IN_27_AID, ADR(in_as[27]));
	inxt(IN_28_AID, ADR(in_as[28]));
	inxt(IN_29_AID, ADR(in_as[29]));
	inxt(IN_30_AID, ADR(in_as[30]));
	inxt(IN_31_AID, ADR(in_as[31]));
	inxt(IN_32_AID, ADR(in_as[32]));
	inxt(IN_33_AID, ADR(in_as[33]));
	inxt(IN_34_AIV,  ADR(in_as[34]));
	inxt(IN_35_AIV, ADR(in_as[35]));
	inxt(IN_36_AIV, ADR(in_as[36]));
	inxt(IN_37_AIV, ADR(in_as[37]));
	inxt(IN_38_AIV, ADR(in_as[38]));
	inxt(IN_52_AIC, ADR(in_as[52]));
	inxt(IN_53_AIC, ADR(in_as[53]));
	inxt(IN_54_AIC, ADR(in_as[54]));
	inxt(IN_55_AIV, ADR(in_as[55]));
	inxt(IN_56_AIC, ADR(in_as[56]));
	inxt(IN_62_AIT, ADR(in_as[62]));

(*------------------------------------------------------------------------------ ACTIONS ------------------------------------------------------------------------------*)

	_2_1_PANEL();
	_2_2_HANDLEBAR();
	_2_3_SENSORS();
END_PROGRAM
ACTION _2_1_PANEL:
(*------------------------------------------------------------------------------ DIGITAL ------------------------------------------------------------------------------*)

	in_Panel_Emegency := in_as[9].in_aiv_s.state_l;
(*	in_Panel_Wireless := in_as[10].in_aiv_s.state_l; *)
(*	in_Panel_Wire := in_as[10].in_aiv_s.state_l; *)
	in_Panel_Manual := in_as[11].in_aiv_s.state_l;
	in_Panel_Heater := in_as[12].in_aiv_s.state_l;
	in_Panel_Engine_On := in_as[13].in_aiv_s.state_l;
	in_Panel_Engine_Off := in_as[14].in_aiv_s.state_l;
	in_Panel_Wheel_Up := in_as[15].in_aiv_s.state_l;;
	in_Panel_Wheel_Down := in_as[16].in_aiv_s.state_l;
	in_Panel_Buzzer_On := in_as[17].in_aiv_s.state_l;
	in_Panel_Buzzer_Off := in_as[18].in_aiv_s.state_l;
	in_Panel_Cyl_Z_Up := in_as[19].in_aiv_s.state_l;
	in_Panel_Cyl_Z_Down := in_as[20].in_aiv_s.state_l;
	in_Panel_Cyl_XY_Up := in_as[21].in_aiv_s.state_l;;
	in_Panel_Cyl_XY_Down := in_as[22].in_aiv_s.state_l;
	in_Panel_X_select := in_as[23].in_aiv_s.state_l;
	in_Panel_Y_select := in_as[24].in_aiv_s.state_l;
	in_Panel_Zero_Return := in_as[28].in_aiv_s.state_l;
	in_Panel_A_select := in_as[43].in_di_s.state_l;
	in_Panel_B_select := in_as[44].in_di_s.state_l;
	in_Panel_C_select := in_as[45].in_di_s.state_l;
	in_Panel_D_select := in_as[46].in_di_s.state_l;
	in_Panel_Group1_select := in_as[47].in_di_s.state_l;
	in_Panel_Group2_select := in_as[48].in_di_s.state_l;

(*------------------------------------------------------------------------------ ANALOG ------------------------------------------------------------------------------*)

	in_Panel_Voltmeter := in_as[55].in_aiv_s.u_mV_u16;
END_ACTION
ACTION _2_2_HANDLEBAR:
(*------------------------------------------------------------------------------ JOYSTICK INPUT ------------------------------------------------------------------------------*)

	in_Handlebar_Joy := INT_TO_DINT(in_as[8].in_aiv_s.u_mV_u16);

(*------------------------------------------------------------------------------CALC_IN ------------------------------------------------------------------------------*)
(*
	Handelbar_Joy_upward := mat_calcScale(in_Handlebar_Joy, Para_s.Handelbar_Joy_Up_Min, Handelbar_Joy_Up_Max, 0, 1000);
	Handelbar_Joy_downward := mat_calcScale(in_Handlebar_Joy, Para_s.Handelbar_Joy_Down_Min, Para_s.Handelbar_Joy_Down_Max, 0, 1000);
*)

(*------------------------------------------------------------------------------WHEEL SENSOR ------------------------------------------------------------------------------*)

	in_Sensor_Wheel_rest := in_as[25].in_aiv_s.state_l;
END_ACTION
ACTION _2_3_SENSORS:
(*------------------------------------------------------------------------------ GEFRAN TWIIST SENSOR INPUT ------------------------------------------------------------------------------*)

	in_Sensor_Distance_X := in_as[52].in_aic_s.i_uA_u16;
	in_Sensor_Distance_Y := in_as[53].in_aic_s.i_uA_u16;
	in_Sensor_Distance_Z := in_as[54].in_aic_s.i_uA_u16;

(*------------------------------------------------------------------------------ GEFRAN PRESSURE SENSOR INPUT ------------------------------------------------------------------------------*)

	in_Sensor_Pressure_X_A := in_as[1].in_aiv_s.u_mV_u16;
	in_Sensor_Pressure_X_B := in_as[2].in_aiv_s.u_mV_u16;
	in_Sensor_Pressure_Y_A := in_as[3].in_aiv_s.u_mV_u16;
	in_Sensor_Pressure_Y_B := in_as[4].in_aiv_s.u_mV_u16;
	in_Sensor_Pressure_Z_A := in_as[5].in_aiv_s.u_mV_u16;
	in_Sensor_Pressure_Z_B := in_as[6].in_aiv_s.u_mV_u16;
	in_Sensor_Pressure_Main := in_as[7].in_aiv_s.u_mV_u16;

(*------------------------------------------------------------------------------ TANK  SENSOR INPUT ------------------------------------------------------------------------------*)

	in_Sensor_Voltage := in_as[55].in_aiv_s.u_mV_u16;

(*------------------------------------------------------------------------------ TANK  SENSOR INPUT ------------------------------------------------------------------------------*)

	in_Sensor_Temp := in_as[62].in_ait_s.t_C_s16;

	in_Sensor_Oil_Low := in_as[29].in_aiv_s.state_l;
	in_Sensor_Oil_Low_Low := in_as[30].in_aiv_s.state_l;
	in_Sensor_Filter_indicator := in_as[31].in_aiv_s.state_l;
	in_Sensor_Temp_High := in_as[32].in_aiv_s.state_l;
	in_Sensor_Overcurrent := in_as[33].in_aiv_s.state_l;
END_ACTION

(* POU _3_RUN, ST *)
PROGRAM _3_RUN
VAR

(* OUTPUT *)
	out_Cyl_X_up: UINT;
	out_Cyl_X_down: UINT;
	out_Cyl_Y_up: UINT;
	out_Cyl_Y_down: UINT;
	out_Cyl_Z_up_load: UINT;
	out_Cyl_Z_down_load: UINT;
	out_Cyl_Z_up_noload: UINT;
	out_Cyl_Z_down_noload: UINT;
	out_Track_forward: UINT;
	out_Track_backward: UINT;
	out_Wheel_up: UINT;
	out_Wheel_down: UINT;
	out_3Way: UINT;
	out_Unloading: UINT;
	out_Buzzer: UINT;
	out_ACmotor_start: UINT;
	out_ACmotor_stop: UINT;
	out_Heater: UINT;
	out_Resist: UINT;

(* Ramp *)
	Ramp_Cyl_X_up: RAMP_INT;
	Ramp_Cyl_X_down: RAMP_INT;
	Ramp_Cyl_Y_up: RAMP_INT;
	Ramp_Cyl_Y_down: RAMP_INT;
	Ramp_Cyl_Z_up: RAMP_INT;
	Ramp_Cyl_Z_down: RAMP_INT;
	Ramp_Track_forward: RAMP_INT;
	Ramp_Track_backward: RAMP_INT;
	Ramp_Wheel_up: RAMP_INT;
	Ramp_Wheel_down: RAMP_INT;

(* Error *)
	Input_Error_Wheel_UpDown: BOOL;
	Input_Error_Engine_OnOff: BOOL;
	Input_Error_Buzzer_OnOff: BOOL;

END_VAR
VAR_INPUT

END_VAR
IF (NOT _2_IN_RC.in_Panel_Manual) AND NOT (_2_IN_RC.) THEN
	_3_1_JOYSTICK_MODE();
ELSIF (in_as[10]) AND NOT (in_as[11]) THEN
	_3_2_MICRO_MODE();
ELSIF (_2_IN_RC.in_Panel_Manual) THEN
	_3_3_ROTATION_MODE();
END_IF;

	_3_4_WHEEL();
	_3_5_TRACK();
	_3_6_ONOFF();
	_3_7_ERROR();
END_PROGRAM
ACTION _3_1_JOYSTICK_MODE:
;
END_ACTION
ACTION _3_2_MICRO_MODE:
;
END_ACTION
ACTION _3_3_ROTATION_MODE:
;
END_ACTION
ACTION _3_4_WHEEL:
(*------------------------------------------------------------------------------ WHEEL UP ------------------------------------------------------------------------------*)

	IF (_2_IN_RC.in_Panel_Wheel_Up) AND NOT(_2_IN_RC.in_Panel_Wheel_Down) THEN
		Ramp_Wheel_up(in:=1000, ASCEND:=, DESCEND:=, TIMEBASE:=, RESET:=FALSE);
(*		out_Wheel_up := DINT_TO_UINT(mat_calcScale(Ramp_Wheel_up.out, 0, 1000, , ); *)

(*------------------------------------------------------------------------------ WHEEL UP ------------------------------------------------------------------------------*)

	ELSIF NOT(_2_IN_RC.in_Panel_Wheel_Up) AND (_2_IN_RC.in_Panel_Wheel_Down) THEN
		Ramp_Wheel_down(in:=1000, ASCEND:=, DESCEND:=, TIMEBASE:=, RESET:=FALSE);
(*		out_Wheel_down := DINT_TO_UINT(mat_calcScale(Ramp_Wheel_down.out, 0, 1000, , ); *)

(*------------------------------------------------------------------------------No mover or Operator Error ------------------------------------------------------------------------------*)

	ELSE
(*		Ramp_Wheel_up(in:=0, ASCEND:=, DESCEND:=, TIMEBASE:=, RESET:=FALSE); *)
		out_Wheel_up := DINT_TO_UINT(mat_calcScale(Ramp_Wheel_up.out, 0, 1000, , );
		Ramp_Wheel_down(in:=0, ASCEND:=, DESCEND:=, TIMEBASE:=, RESET:=FALSE);
(*		out_Wheel_down := DINT_TO_UINT(mat_calcScale(Ramp_Wheel_down.out, 0, 1000, , ); *)

	END_IF;
END_ACTION
ACTION _3_5_TRACK:
(*------------------------------------------------------------------------------ TRACK forward / backward ------------------------------------------------------------------------------*)


IF NOT (_2_IN_RC.in_Sensor_Wheel_rest) THEN

(*
	Ramp_Track_forward(in:=_2_IN_RC.Handelbar_Joy_upward, ASCED:=, DESECND:=, TIMEBASE:=, RESET:=FALSE);
	out_Track_forward := DINT_TO_UINT(mat_calcScale(Ramp_Track_forward.out, 0, 1000, , ));

	Ramp_Track_backward(in:=_2_IN_RC.Handelbar_Joy_downward, ASCED:=, DESECND:=, TIMEBASE:=, RESET:=FALSE);
	out_Track_backward := DINT_TO_UINT(mat_calcScale(Ramp_Track_backward.out, 0, 1000, , ));
*)
	out_Wheel_up := 0;
	out_Wheel_down := 0;

(*------------------------------------------------------------------------------ Track Stop ------------------------------------------------------------------------------*)

ELSE

	out_Track_forward := 0;
	out_Track_backward := 0;

END_IF;
END_ACTION
ACTION _3_6_ONOFF:
(*------------------------------------------------------------------------------ Buzzer On / Off ------------------------------------------------------------------------------*)

IF (Input_Error_Buzzer_OnOff) THEN
	out_Buzzer := 0;
ELSE

	(* Conditions for Buzzer On -> add *)

	IF  (_3_RUN.in_Panel_Buzzer_Off) THEN
		out_Buzzer := 0;
	ELSIF (_3_RUN.in_Panel_Buzzer_On) THEN
		out_Buzzer := 1;
(*	ELSE
		out_Buzzer := 0; *)
	END_IF;

END_IF;

(*------------------------------------------------------------------------------ Engine Start / Stop ------------------------------------------------------------------------------*)

IF (_3_RUN.in_Panel_Engine_Off) THEN
	out_ACmotor_stop := 1;
ELSE
	out_ACmotor_stop := 0;
END_IF;

IF (_3_RUN.in_Panel_Engine_On) THEN
	out_ACmotor_start := 1;
ELSE
	out_ACmotor_start := 0;
END_IF;
END_ACTION
ACTION _3_7_ERROR:
(*------------------------------------------------------------------------------ Alert 1 ------------------------------------------------------------------------------*)

(*------------------------------------------------------------------------------ Alert 1 ------------------------------------------------------------------------------*)

(*------------------------------------------------------------------------------ Alert 3 : Operator Error ------------------------------------------------------------------------------*)

(* Engine On/Off double Input Error *)

IF (_3_RUN.in_Panel_Engine_On) AND (_3_RUN.in_Panel_Engine_Off) THEN
	Input_Error_Engine_OnOff := TRUE;
ELSE
	Input_Error_Engine_OnOff := FALSE;
END_IF;

(* Wheel Up/Down double Input Error *)

IF (_3_RUN.in_Panel_Wheel_Up) AND (_3_RUN.in_Panel_Wheel_Down) THEN
	Input_Error_Wheel_UpDown := TRUE;
ELSE
	Input_Error_Wheel_UpDown := FALSE;
END_IF;


(* Buzzer On/Off double Input Error *)

IF (_3_RUN.in_Panel_Buzzer_On) AND (_3_RUN.in_Panel_Buzzer_Off) THEN
	Input_Error_Buzzer_OnOff := TRUE;
ELSE
	Input_Error_Buzzer_OnOff := FALSE;
END_IF;
END_ACTION

(* POU _4_PROCESS_VALUES, ST *)
PROGRAM _4_PROCESS_VALUES
VAR
END_VAR
;
END_PROGRAM

(* POU _5_OUT_RC, ST *)
PROGRAM _5_OUT_RC
VAR
	out_as: ARRAY [1..73] OF out_ts;
END_VAR
IF (_2_IN_RC.in_Panel_Emegency) THEN

(*------------------------------------------------------------------------------ 1. Emergency Mode ------------------------------------------------------------------------------*)

(* Propotional Output*)
	out(OUT_1_POH, 0);
	out(OUT_2_POH, 0);
	out(OUT_3_POH, 0);
	out(OUT_4_POH, 0);
	out(OUT_5_POH, 0);
	out(OUT_6_POH, 0);
	out(OUT_7_POH, 0);
	out(OUT_8_POH, 0);
	out(OUT_9_POH, 0);
	out(OUT_10_POH, 0);
	out(OUT_37_POL, 0);
	out(OUT_38_POL, 0);

(* Digital Output*)
	out(OUT_19_DOH, 0);
	out(OUT_20_DOH, 0);
	out(OUT_21_DOH, 0);
	out(OUT_22_DOH, 0);
	out(OUT_23_DOH, 0);
	out(OUT_24_DOH, 0);
	out(OUT_25_DOH, 0);

(*------------------------------------------------------------------------------ 2. Normal Mode ------------------------------------------------------------------------------*)

ELSE

	out(OUT_1_POH, _3_RUN.out_Cyl_X_up);
	out(OUT_2_POH, _3_RUN.out_Cyl_X_down);
	out(OUT_3_POH, _3_RUN.out_Cyl_Y_up);
	out(OUT_4_POH, _3_RUN.out_Cyl_Y_down);
	out(OUT_5_POH, _3_RUN.out_Cyl_Z_up_noload);
	out(OUT_6_POH, _3_RUN.out_Cyl_Z_down_noload);
	out(OUT_7_POH, _3_RUN.out_Cyl_Z_up_load);
	out(OUT_8_POH, _3_RUN.out_Cyl_Z_down_load);
	out(OUT_9_POH, _3_RUN.out_Track_forward);
	out(OUT_10_POH, _3_RUN.out_Track_backward);
	out(OUT_37_POL, _3_RUN.out_Wheel_up);
	out(OUT_38_POL, _3_RUN.out_Wheel_down);

	out(OUT_19_DOH, _3_RUN.out_3Way);
	out(OUT_20_DOH, _3_RUN.out_Unloading);
	out(OUT_21_DOH, _3_RUN.out_Buzzer);
	out(OUT_22_DOH, _3_RUN.out_ACmotor_start);
	out(OUT_23_DOH, _3_RUN.out_ACmotor_stop);
	out(OUT_24_DOH, _3_RUN.out_Heater);
	out(OUT_25_DOH, _3_RUN.out_Resist);

END_IF;
END_PROGRAM
ACTION _5_1_OUT_STATUS:
(*** Output Status ***)

(** Propotional Valve **)

 out_getStatusxt(OUT_1_POH, ADR(out_as[1]));			(* Cyline X Up *)
 out_getStatusxt(OUT_2_POH, ADR(out_as[2]));			(* Cyline X Down *)
 out_getStatusxt(OUT_3_POH, ADR(out_as[3]));			(* Cyline Y Up *)
 out_getStatusxt(OUT_4_POH, ADR(out_as[4]));			(* Cyline Y Down *)
 out_getStatusxt(OUT_5_POH, ADR(out_as[5]));			(* Cyline Z Up with Load *)
 out_getStatusxt(OUT_6_POH, ADR(out_as[6]));			(* Cyline Z Down with Load *)
 out_getStatusxt(OUT_7_POH, ADR(out_as[7]));			(* Cyline Z Up without Load *)
 out_getStatusxt(OUT_8_POH, ADR(out_as[8]));			(* Cyline Z Down without Load *)
 out_getStatusxt(OUT_37_POL, ADR(out_as[37]));		(* Cyline X Up *)
 out_getStatusxt(OUT_38_POL, ADR(out_as[38]));		(* Cyline X Up *)

(** On/Off **)

 out_getStatusxt(OUT_19_DOH, ADR(out_as[21]));		(* 3-way Sol <- load/noload change *)
 out_getStatusxt(OUT_20_DOH, ADR(out_as[22]));		(* Unloading Sol <- NO, alway on to create pressure *)
 out_getStatusxt(OUT_21_DOH, ADR(out_as[21]));		(* Buzzer *)
 out_getStatusxt(OUT_22_DOH, ADR(out_as[22]));		(* Engine Start *)
 out_getStatusxt(OUT_23_DOH, ADR(out_as[23]));		(* Engine Stop *)
 out_getStatusxt(OUT_24_DOH, ADR(out_as[24]));		(* Heater ON *)
 out_getStatusxt(OUT_25_DOH, ADR(out_as[25]));		(* Teminal Resistance *)
END_ACTION

(* POU Autocode/Callback_diag_getPara, ST *)
PROGRAM Callback_diag_getPara
VAR
   eep:  ARRAY [0..3840] OF INT;
END_VAR
(*********************************************)
(*  DON'T MAKE ANY CHANGES TO THIS PROGRAM!! *)
(*     FILE WAS AUTOMATICALLY GENERATED!!    *)
(*********************************************)

(* get EEPROM pages 0..14 *)
ree_getArray( PAGE0,  0, ADR(eep[0]),    256 );
ree_getArray( PAGE1,  0, ADR(eep[256]),  256 );
ree_getArray( PAGE2,  0, ADR(eep[512]),  256 );
ree_getArray( PAGE3,  0, ADR(eep[768]),  256 );
ree_getArray( PAGE4,  0, ADR(eep[1024]), 256 );
ree_getArray( PAGE5,  0, ADR(eep[1280]), 256 );
ree_getArray( PAGE6,  0, ADR(eep[1536]), 256 );
ree_getArray( PAGE7,  0, ADR(eep[1792]), 256 );
ree_getArray( PAGE8,  0, ADR(eep[2048]), 256 );
ree_getArray( PAGE9,  0, ADR(eep[2304]), 256 );
ree_getArray( PAGE10, 0, ADR(eep[2560]), 256 );
ree_getArray( PAGE11, 0, ADR(eep[2816]), 256 );
ree_getArray( PAGE12, 0, ADR(eep[3072]), 256 );
ree_getArray( PAGE13, 0, ADR(eep[3328]), 256 );
ree_getArray( PAGE14, 0, ADR(eep[3584]), 256 );


(* Input configuration *)

(* Joystick 12 Min Max *)
    para_s.L1_Joy_Up_Min_s16                  := eep[EEP_L1_Joy_Up_Min_e];
    para_s.L1_Joy_Up_Max_s16                  := eep[EEP_L1_Joy_Up_Max_e];
    para_s.L1_Joy_Down_Min_s16                := eep[EEP_L1_Joy_Down_Min_e];
    para_s.L1_Joy_Down_Max_s16                := eep[EEP_L1_Joy_Down_Max_e];
    para_s.L2_Joy_Up_Min_s16                  := eep[EEP_L2_Joy_Up_Min_e];
    para_s.L2_Joy_Up_Max_s16                  := eep[EEP_L2_Joy_Up_Max_e];
    para_s.L2_Joy_Down_Min_s16                := eep[EEP_L2_Joy_Down_Min_e];
    para_s.L2_Joy_Down_Max_s16                := eep[EEP_L2_Joy_Down_Max_e];

(* Joystick 34 Min Max *)
    para_s.L3_Joy_Up_Min_s16                  := eep[EEP_L3_Joy_Up_Min_e];
    para_s.L3_Joy_Up_Max_s16                  := eep[EEP_L3_Joy_Up_Max_e];
    para_s.L3_Joy_Down_Min_s16                := eep[EEP_L3_Joy_Down_Min_e];
    para_s.L3_Joy_Down_Max_s16                := eep[EEP_L3_Joy_Down_Max_e];
    para_s.L4_Joy_Up_Min_s16                  := eep[EEP_L4_Joy_Up_Min_e];
    para_s.L4_Joy_Up_Max_s16                  := eep[EEP_L4_Joy_Up_Max_e];
    para_s.L4_Joy_Down_Min_s16                := eep[EEP_L4_Joy_Down_Min_e];
    para_s.L4_Joy_Down_Max_s16                := eep[EEP_L4_Joy_Down_Max_e];

(* Joystick Master Min Max *)
    para_s.M_Joy_Up_Min_s16                   := eep[EEP_M_Joy_Up_Min_e];
    para_s.M_Joy_Up_Max_s16                   := eep[EEP_M_Joy_Up_Max_e];
    para_s.M_Joy_Down_Min_s16                 := eep[EEP_M_Joy_Down_Min_e];
    para_s.M_Joy_Down_Max_s16                 := eep[EEP_M_Joy_Down_Max_e];

(* Pump 12 Current Control *)
    para_s.iPump_PV1A_min_s16                 := eep[EEP_iPump_PV1A_min_e];
    para_s.iPump_PV1A_max_s16                 := eep[EEP_iPump_PV1A_max_e];
    para_s.iPump_PV1B_min_s16                 := eep[EEP_iPump_PV1B_min_e];
    para_s.iPump_PV1B_max_s16                 := eep[EEP_iPump_PV1B_max_e];
    para_s.iPump_PV2A_min_s16                 := eep[EEP_iPump_PV2A_min_e];
    para_s.iPump_PV2A_max_s16                 := eep[EEP_iPump_PV2A_max_e];
    para_s.iPump_PV2B_min_s16                 := eep[EEP_iPump_PV2B_min_e];
    para_s.iPump_PV2B_max_s16                 := eep[EEP_iPump_PV2B_max_e];

(* Pump 34 Current Control *)
    para_s.iPump_PV3A_min_s16                 := eep[EEP_iPump_PV3A_min_e];
    para_s.iPump_PV3A_max_s16                 := eep[EEP_iPump_PV3A_max_e];
    para_s.iPump_PV3B_min_s16                 := eep[EEP_iPump_PV3B_min_e];
    para_s.iPump_PV3B_max_s16                 := eep[EEP_iPump_PV3B_max_e];
    para_s.iPump_PV4A_min_s16                 := eep[EEP_iPump_PV4A_min_e];
    para_s.iPump_PV4A_max_s16                 := eep[EEP_iPump_PV4A_max_e];
    para_s.iPump_PV4B_min_s16                 := eep[EEP_iPump_PV4B_min_e];
    para_s.iPump_PV4B_max_s16                 := eep[EEP_iPump_PV4B_max_e];

(* Pump 56 Current Control *)
    para_s.iPump_PV5A_min_s16                 := eep[EEP_iPump_PV5A_min_e];
    para_s.iPump_PV5A_max_s16                 := eep[EEP_iPump_PV5A_max_e];
    para_s.iPump_PV5B_min_s16                 := eep[EEP_iPump_PV5B_min_e];
    para_s.iPump_PV5B_max_s16                 := eep[EEP_iPump_PV5B_max_e];
    para_s.iPump_PV6A_min_s16                 := eep[EEP_iPump_PV6A_min_e];
    para_s.iPump_PV6A_max_s16                 := eep[EEP_iPump_PV6A_max_e];
    para_s.iPump_PV6B_min_s16                 := eep[EEP_iPump_PV6B_min_e];
    para_s.iPump_PV6B_max_s16                 := eep[EEP_iPump_PV6B_max_e];

(* Pump 78 Current Control *)
    para_s.iPump_PV7A_min_s16                 := eep[EEP_iPump_PV7A_min_e];
    para_s.iPump_PV7A_max_s16                 := eep[EEP_iPump_PV7A_max_e];
    para_s.iPump_PV7B_min_s16                 := eep[EEP_iPump_PV7B_min_e];
    para_s.iPump_PV7B_max_s16                 := eep[EEP_iPump_PV7B_max_e];
    para_s.iPump_PV8A_min_s16                 := eep[EEP_iPump_PV8A_min_e];
    para_s.iPump_PV8A_max_s16                 := eep[EEP_iPump_PV8A_max_e];
    para_s.iPump_PV8B_min_s16                 := eep[EEP_iPump_PV8B_min_e];
    para_s.iPump_PV8B_max_s16                 := eep[EEP_iPump_PV8B_max_e];

(* Local Pump Current Control *)
    para_s.iPump_Local_PV15A_max_s16          := eep[EEP_iPump_Local_PV15A_max_e];
    para_s.iPump_Local_PV26A_max_s16          := eep[EEP_iPump_Local_PV26A_max_e];
    para_s.iPump_Local_PV37A_max_s16          := eep[EEP_iPump_Local_PV37A_max_e];
    para_s.iPump_Local_PV48A_max_s16          := eep[EEP_iPump_Local_PV48A_max_e];
    para_s.iPump_Local_PV15B_max_s16          := eep[EEP_iPump_Local_PV15B_max_e];
    para_s.iPump_Local_PV26B_max_s16          := eep[EEP_iPump_Local_PV26B_max_e];
    para_s.iPump_Local_PV37B_max_s16          := eep[EEP_iPump_Local_PV37B_max_e];
    para_s.iPump_Local_PV48B_max_s16          := eep[EEP_iPump_Local_PV48B_max_e];


(* Input configuration 2 *)

(* Ramp_PV1AB *)
    para_s.Ramp_PV1A_Ascend_s16               := eep[EEP_Ramp_PV1A_Ascend_e];
    para_s.Ramp_PV1A_Descend_s16              := eep[EEP_Ramp_PV1A_Descend_e];
    para_s.Ramp_PV1A_Timebase_s16             := eep[EEP_Ramp_PV1A_Timebase_e];
    para_s.Ramp_PV1B_Ascend_s16               := eep[EEP_Ramp_PV1B_Ascend_e];
    para_s.Ramp_PV1B_Descend_s16              := eep[EEP_Ramp_PV1B_Descend_e];
    para_s.Ramp_PV1B_Timebase_s16             := eep[EEP_Ramp_PV1B_Timebase_e];

(* Ramp_PV2AB *)
    para_s.Ramp_PV2A_Ascend_s16               := eep[EEP_Ramp_PV2A_Ascend_e];
    para_s.Ramp_PV2A_Descend_s16              := eep[EEP_Ramp_PV2A_Descend_e];
    para_s.Ramp_PV2A_Timebase_s16             := eep[EEP_Ramp_PV2A_Timebase_e];
    para_s.Ramp_PV2B_Ascend_s16               := eep[EEP_Ramp_PV2B_Ascend_e];
    para_s.Ramp_PV2B_Descend_s16              := eep[EEP_Ramp_PV2B_Descend_e];
    para_s.Ramp_PV2B_Timebase_s16             := eep[EEP_Ramp_PV2B_Timebase_e];

(* Ramp_PV3AB *)
    para_s.Ramp_PV3A_Ascend_s16               := eep[EEP_Ramp_PV3A_Ascend_e];
    para_s.Ramp_PV3A_Descend_s16              := eep[EEP_Ramp_PV3A_Descend_e];
    para_s.Ramp_PV3A_Timebase_s16             := eep[EEP_Ramp_PV3A_Timebase_e];
    para_s.Ramp_PV3B_Ascend_s16               := eep[EEP_Ramp_PV3B_Ascend_e];
    para_s.Ramp_PV3B_Descend_s16              := eep[EEP_Ramp_PV3B_Descend_e];
    para_s.Ramp_PV3B_Timebase_s16             := eep[EEP_Ramp_PV3B_Timebase_e];

(* Ramp_PV4AB *)
    para_s.Ramp_PV4A_Ascend_s16               := eep[EEP_Ramp_PV4A_Ascend_e];
    para_s.Ramp_PV4A_Descend_s16              := eep[EEP_Ramp_PV4A_Descend_e];
    para_s.Ramp_PV4A_Timebase_s16             := eep[EEP_Ramp_PV4A_Timebase_e];
    para_s.Ramp_PV4B_Ascend_s16               := eep[EEP_Ramp_PV4B_Ascend_e];
    para_s.Ramp_PV4B_Descend_s16              := eep[EEP_Ramp_PV4B_Descend_e];
    para_s.Ramp_PV4B_Timebase_s16             := eep[EEP_Ramp_PV4B_Timebase_e];

(* Ramp_PV5AB *)
    para_s.Ramp_PV5A_Ascend_s16               := eep[EEP_Ramp_PV5A_Ascend_e];
    para_s.Ramp_PV5A_Descend_s16              := eep[EEP_Ramp_PV5A_Descend_e];
    para_s.Ramp_PV5A_Timebase_s16             := eep[EEP_Ramp_PV5A_Timebase_e];
    para_s.Ramp_PV5B_Ascend_s16               := eep[EEP_Ramp_PV5B_Ascend_e];
    para_s.Ramp_PV5B_Descend_s16              := eep[EEP_Ramp_PV5B_Descend_e];
    para_s.Ramp_PV5B_Timebase_s16             := eep[EEP_Ramp_PV5B_Timebase_e];

(* Ramp_PV6AB *)
    para_s.Ramp_PV6A_Ascend_s16               := eep[EEP_Ramp_PV6A_Ascend_e];
    para_s.Ramp_PV6A_Descend_s16              := eep[EEP_Ramp_PV6A_Descend_e];
    para_s.Ramp_PV6A_Timebase_s16             := eep[EEP_Ramp_PV6A_Timebase_e];
    para_s.Ramp_PV6B_Ascend_s16               := eep[EEP_Ramp_PV6B_Ascend_e];
    para_s.Ramp_PV6B_Descend_s16              := eep[EEP_Ramp_PV6B_Descend_e];
    para_s.Ramp_PV6B_Timebase_s16             := eep[EEP_Ramp_PV6B_Timebase_e];

(* Ramp_PV7AB *)
    para_s.Ramp_PV7A_Ascend_s16               := eep[EEP_Ramp_PV7A_Ascend_e];
    para_s.Ramp_PV7A_Descend_s16              := eep[EEP_Ramp_PV7A_Descend_e];
    para_s.Ramp_PV7A_Timebase_s16             := eep[EEP_Ramp_PV7A_Timebase_e];
    para_s.Ramp_PV7B_Ascend_s16               := eep[EEP_Ramp_PV7B_Ascend_e];
    para_s.Ramp_PV7B_Descend_s16              := eep[EEP_Ramp_PV7B_Descend_e];
    para_s.Ramp_PV7B_Timebase_s16             := eep[EEP_Ramp_PV7B_Timebase_e];

(* Ramp_PV8AB *)
    para_s.Ramp_PV8A_Ascend_s16               := eep[EEP_Ramp_PV8A_Ascend_e];
    para_s.Ramp_PV8A_Descend_s16              := eep[EEP_Ramp_PV8A_Descend_e];
    para_s.Ramp_PV8A_Timebase_s16             := eep[EEP_Ramp_PV8A_Timebase_e];
    para_s.Ramp_PV8B_Ascend_s16               := eep[EEP_Ramp_PV8B_Ascend_e];
    para_s.Ramp_PV8B_Descend_s16              := eep[EEP_Ramp_PV8B_Descend_e];
    para_s.Ramp_PV8B_Timebase_s16             := eep[EEP_Ramp_PV8B_Timebase_e];


(* Input configuration 3 *)

(* Ramp_PV_Local *)
    para_s.Ramp_PV_Local_Ascend_s16           := eep[EEP_Ramp_PV_Local_Ascend_e];
    para_s.Ramp_PV_Local_Descend_s16          := eep[EEP_Ramp_PV_Local_Descend_e];
    para_s.Ramp_PV_Local_Timebase_s16         := eep[EEP_Ramp_PV_Local_Timebase_e];

(* AutoLeveling_height *)
    para_s.Max_height_2_s16                   := eep[EEP_Max_height_2_e];
    para_s.Max_height_3_s16                   := eep[EEP_Max_height_3_e];
    para_s.Max_height_4_s16                   := eep[EEP_Max_height_4_e];
    para_s.Min_height_2_s16                   := eep[EEP_Min_height_2_e];
    para_s.Min_height_3_s16                   := eep[EEP_Min_height_3_e];
    para_s.Min_height_4_s16                   := eep[EEP_Min_height_4_e];

(* AutoLeveling_PV *)
    para_s.AutoLeveling_compensator_1_s16     := eep[EEP_AutoLeveling_compensator_1_e];
    para_s.AutoLeveling_compensator_2_up_s16  := eep[EEP_AutoLeveling_compensator_2_up_e];
    para_s.AutoLeveling_compensator_2_down_s16 := eep[EEP_AutoLeveling_compensator_2_down_e];
    para_s.AutoLeveling_compensator_3_up_s16  := eep[EEP_AutoLeveling_compensator_3_up_e];
    para_s.AutoLeveling_compensator_3_down_s16 := eep[EEP_AutoLeveling_compensator_3_down_e];
    para_s.AutoLeveling_compensator_4_up_s16  := eep[EEP_AutoLeveling_compensator_4_up_e];
    para_s.AutoLeveling_compensator_4_down_s16 := eep[EEP_AutoLeveling_compensator_4_down_e];

(* Distance *)
    para_s.Distance_1_to_4_s16                := eep[EEP_Distance_1_to_4_e];
    para_s.Distance_1_to_2_s16                := eep[EEP_Distance_1_to_2_e];
    para_s.Height_Hysteresis_High_s16         := eep[EEP_Height_Hysteresis_High_e];
    para_s.Height_Hysteresis_Low_s16          := eep[EEP_Height_Hysteresis_Low_e];

(* Height_diff_1 *)
    para_s.Height_diff_point_plus_1_s16       := eep[EEP_Height_diff_point_plus_1_e];
    para_s.Height_diff_point_plus_2_s16       := eep[EEP_Height_diff_point_plus_2_e];
    para_s.Height_diff_point_plus_3_s16       := eep[EEP_Height_diff_point_plus_3_e];
    para_s.Height_diff_point_plus_4_s16       := eep[EEP_Height_diff_point_plus_4_e];
    para_s.Height_diff_point_plus_5_s16       := eep[EEP_Height_diff_point_plus_5_e];
    para_s.Height_diff_point_plus_6_s16       := eep[EEP_Height_diff_point_plus_6_e];
    para_s.Height_diff_point_plus_7_s16       := eep[EEP_Height_diff_point_plus_7_e];
    para_s.Height_diff_point_plus_8_s16       := eep[EEP_Height_diff_point_plus_8_e];

(* Height_diff_2 *)
    para_s.Height_diff_point_minus_1_s16      := eep[EEP_Height_diff_point_minus_1_e];
    para_s.Height_diff_point_minus_2_s16      := eep[EEP_Height_diff_point_minus_2_e];
    para_s.Height_diff_point_minus_3_s16      := eep[EEP_Height_diff_point_minus_3_e];
    para_s.Height_diff_point_minus_4_s16      := eep[EEP_Height_diff_point_minus_4_e];
    para_s.Height_diff_point_minus_5_s16      := eep[EEP_Height_diff_point_minus_5_e];
    para_s.Height_diff_point_minus_6_s16      := eep[EEP_Height_diff_point_minus_6_e];
    para_s.Height_diff_point_minus_7_s16      := eep[EEP_Height_diff_point_minus_7_e];
    para_s.Height_diff_point_minus_8_s16      := eep[EEP_Height_diff_point_minus_8_e];


(* Distance_diff *)

(* Autoset_Phase *)
    para_s.Autoset_PV_phase_1_s16             := eep[EEP_Autoset_PV_phase_1_e];
    para_s.Autoset_PV_phase_2_s16             := eep[EEP_Autoset_PV_phase_2_e];
    para_s.Autoset_PV_phase_3_s16             := eep[EEP_Autoset_PV_phase_3_e];
    para_s.Autoset_PV_phase_4_s16             := eep[EEP_Autoset_PV_phase_4_e];
    para_s.Autoset_PV_phase_5_s16             := eep[EEP_Autoset_PV_phase_5_e];
    para_s.AutoLeveling_PV_phase_0_s16        := eep[EEP_AutoLeveling_PV_phase_0_e];

(* Autoleveling_Phase_1 *)
    para_s.AutoLeveling_PV_phase_1_s16        := eep[EEP_AutoLeveling_PV_phase_1_e];
    para_s.AutoLeveling_PV_phase_2_s16        := eep[EEP_AutoLeveling_PV_phase_2_e];
    para_s.AutoLeveling_PV_phase_3_s16        := eep[EEP_AutoLeveling_PV_phase_3_e];
    para_s.AutoLeveling_PV_phase_4_s16        := eep[EEP_AutoLeveling_PV_phase_4_e];
    para_s.AutoLeveling_PV_phase_5_s16        := eep[EEP_AutoLeveling_PV_phase_5_e];
    para_s.AutoLeveling_PV_phase_6_s16        := eep[EEP_AutoLeveling_PV_phase_6_e];
    para_s.AutoLeveling_PV_phase_7_s16        := eep[EEP_AutoLeveling_PV_phase_7_e];
    para_s.AutoLeveling_PV_phase_8_s16        := eep[EEP_AutoLeveling_PV_phase_8_e];

(* Autoleveling_Phase_2 *)
    para_s.AutoLeveling_PV_phase_9_s16        := eep[EEP_AutoLeveling_PV_phase_9_e];
    para_s.AutoLeveling_PV_phase_10_s16       := eep[EEP_AutoLeveling_PV_phase_10_e];
    para_s.AutoLeveling_PV_phase_11_s16       := eep[EEP_AutoLeveling_PV_phase_11_e];
    para_s.AutoLeveling_PV_phase_12_s16       := eep[EEP_AutoLeveling_PV_phase_12_e];
    para_s.AutoLeveling_PV_phase_13_s16       := eep[EEP_AutoLeveling_PV_phase_13_e];
    para_s.AutoLeveling_PV_phase_14_s16       := eep[EEP_AutoLeveling_PV_phase_14_e];
    para_s.AutoLeveling_PV_phase_15_s16       := eep[EEP_AutoLeveling_PV_phase_15_e];
    para_s.AutoLeveling_PV_phase_16_s16       := eep[EEP_AutoLeveling_PV_phase_16_e];
END_PROGRAM

(* POU _6_CAN_OUT, FBD *)
PROGRAM _6_CAN_OUT
VAR
END_VAR
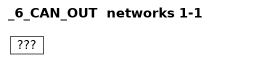
_FBD_ (* Function Block Diagram *)
NETWORK 1
	???
_END_FBD_
(* the same logic as Structured Text *)
(* Network 1 *)
END_PROGRAM
